LIN {X 0,Y 353.263,Z 401.913,A -85,B 0,C 180,E1 -13410,E2 -13410} C_VEL
LIN {X 0,Y 353.204,Z 401.841,A -85,B 0,C 180,E1 -13411.14,E2 -13411.14} C_VEL
LIN {X 0,Y 353.173,Z 401.369,A -85,B 0,C 180,E1 -13412.281,E2 -13412.281} C_VEL
LIN {X 0,Y 353.22,Z 400.459,A -85,B 0,C 180,E1 -13413.422,E2 -13413.422} C_VEL
LIN {X 0,Y 353.263,Z 399.147,A -85,B 0,C 180,E1 -13414.564,E2 -13414.564} C_VEL
LIN {X 0,Y 353.279,Z 397.099,A -85,B 0,C 180,E1 -13415.904,E2 -13415.904} C_VEL
LIN {X 0,Y 353.627,Z 392.597,A -85,B 0,C 180,E1 -13417.997,E2 -13417.997} C_VEL
LIN {X 0,Y 354.079,Z 387.694,A -85,B 0,C 180,E1 -13419.713,E2 -13419.713} C_VEL
LIN {X 0,Y 354.749,Z 381.546,A -85,B 0,C 180,E1 -13421.426,E2 -13421.426} C_VEL
LIN {X 0,Y 355.822,Z 373.938,A -85,B 0,C 180,E1 -13423.128,E2 -13423.128} C_VEL
LIN {X 0,Y 356.761,Z 366.198,A -85,B 0,C 180,E1 -13424.546,E2 -13424.546} C_VEL
LIN {X 0,Y 357.799,Z 356.811,A -85,B 0,C 180,E1 -13425.961,E2 -13425.961} C_VEL
LIN {X 0,Y 359.249,Z 345.191,A -85,B 0,C 180,E1 -13427.357,E2 -13427.357} C_VEL
LIN {X 0,Y 360.513,Z 333.695,A -85,B 0,C 180,E1 -13428.446,E2 -13428.446} C_VEL
LIN {X 0,Y 359.704,Z 322.357,A -85,B 0,C 180,E1 -13429.399,E2 -13429.399} C_VEL
LIN {X 0,Y 357.526,Z 309.013,A -85,B 0,C 180,E1 -13430.353,E2 -13430.353} C_VEL
LIN {X 0,Y 354.606,Z 296.916,A -85,B 0,C 180,E1 -13431.079,E2 -13431.079} C_VEL
LIN {X 0,Y 354.186,Z 294.731,A -85,B 0,C 180,E1 -13431.197,E2 -13431.197} C_VEL
LIN {X 0,Y 354.608,Z 288.932,A -85,B 0,C 180,E1 -13434.594,E2 -13434.594} C_VEL
LIN {X 0,Y 355.173,Z 282.758,A -85,B 0,C 180,E1 -13438.352,E2 -13438.352} C_VEL
LIN {X 0,Y 355.914,Z 276.694,A -85,B 0,C 180,E1 -13442.218,E2 -13442.218} C_VEL
LIN {X 0,Y 356.302,Z 272.736,A -85,B 0,C 180,E1 -13444.89,E2 -13444.89} C_VEL
LIN {X 0,Y 356.369,Z 270.793,A -85,B 0,C 180,E1 -13446.272,E2 -13446.272} C_VEL
LIN {X 0,Y 356.049,Z 266.987,A -85,B 0,C 180,E1 -13449.17,E2 -13449.17} C_VEL
LIN {X 0,Y 355.535,Z 263.321,A -85,B 0,C 180,E1 -13452.227,E2 -13452.227} C_VEL
LIN {X 0,Y 354.835,Z 259.51,A -85,B 0,C 180,E1 -13455.788,E2 -13455.788} C_VEL
LIN {X 0,Y 354.816,Z 259.293,A -85,B 0,C 180,E1 -13458.822,E2 -13458.822} C_VEL
LIN {X 0,Y 354.808,Z 259.292,A -85,B 0,C 180,E1 -13462.401,E2 -13462.401} C_VEL
LIN {X 0,Y 354.81,Z 259.29,A -85,B 0,C 180,E1 -13464.939,E2 -13464.939} C_VEL
LIN {X 0,Y 354.791,Z 259.293,A -85,B 0,C 180,E1 -13468.404,E2 -13468.404} C_VEL
LIN {X 0,Y 354.851,Z 259.284,A -85,B 0,C 180,E1 -13471.618,E2 -13471.618} C_VEL
LIN {X 0,Y 354.896,Z 259.28,A -85,B 0,C 180,E1 -13474.171,E2 -13474.171} C_VEL
LIN {X 0,Y 354.831,Z 259.288,A -85,B 0,C 180,E1 -13477.892,E2 -13477.892} C_VEL
LIN {X 0,Y 354.918,Z 259.277,A -85,B 0,C 180,E1 -13481.89,E2 -13481.89} C_VEL
LIN {X 0,Y 354.937,Z 259.275,A -85,B 0,C 180,E1 -13485.98,E2 -13485.98} C_VEL
LIN {X 0,Y 354.972,Z 259.27,A -85,B 0,C 180,E1 -13489.734,E2 -13489.734} C_VEL
LIN {X 0,Y 355.108,Z 259.254,A -85,B 0,C 180,E1 -13492.035,E2 -13492.035} C_VEL
LIN {X 0,Y 355.086,Z 259.255,A -85,B 0,C 180,E1 -13494.319,E2 -13494.319} C_VEL
LIN {X 0,Y 355.239,Z 259.237,A -85,B 0,C 180,E1 -13497.731,E2 -13497.731} C_VEL
LIN {X 0,Y 355.39,Z 259.217,A -85,B 0,C 180,E1 -13499.999,E2 -13499.999} C_VEL
LIN {X 0,Y 355.239,Z 259.238,A -85,B 0,C 180,E1 -13502.266,E2 -13502.266} C_VEL
LIN {X 0,Y 355.086,Z 259.257,A -85,B 0,C 180,E1 -13505.678,E2 -13505.678} C_VEL
LIN {X 0,Y 355.318,Z 260.942,A -85,B 0,C 180,E1 -13507.957,E2 -13507.957} C_VEL
LIN {X 0,Y 355.247,Z 264.154,A -85,B 0,C 180,E1 -13511.409,E2 -13511.409} C_VEL
LIN {X 0,Y 355.037,Z 266.823,A -85,B 0,C 180,E1 -13514.084,E2 -13514.084} C_VEL
LIN {X 0,Y 354.65,Z 270.896,A -85,B 0,C 180,E1 -13517.977,E2 -13517.977} C_VEL
LIN {X 0,Y 354.303,Z 274.435,A -85,B 0,C 180,E1 -13521.208,E2 -13521.208} C_VEL
LIN {X 0,Y 354.018,Z 278.57,A -85,B 0,C 180,E1 -13524.872,E2 -13524.872} C_VEL
LIN {X 0,Y 358.353,Z 293.464,A -85,B 0,C 180,E1 -13525.871,E2 -13525.871} C_VEL
LIN {X 0,Y 360.827,Z 304.889,A -85,B 0,C 180,E1 -13526.769,E2 -13526.769} C_VEL
LIN {X 0,Y 361.556,Z 309.621,A -85,B 0,C 180,E1 -13527.179,E2 -13527.179} C_VEL
LIN {X 0,Y 360.633,Z 320.768,A -85,B 0,C 180,E1 -13528.128,E2 -13528.128} C_VEL
LIN {X 0,Y 359.465,Z 331.353,A -85,B 0,C 180,E1 -13529.259,E2 -13529.259} C_VEL
LIN {X 0,Y 358.198,Z 341.935,A -85,B 0,C 180,E1 -13530.671,E2 -13530.671} C_VEL
LIN {X 0,Y 357.012,Z 351.025,A -85,B 0,C 180,E1 -13532.171,E2 -13532.171} C_VEL
LIN {X 0,Y 355.829,Z 359.612,A -85,B 0,C 180,E1 -13533.95,E2 -13533.95} C_VEL
LIN {X 0,Y 354.944,Z 366.442,A -85,B 0,C 180,E1 -13535.729,E2 -13535.729} C_VEL
LIN {X 0,Y 354.256,Z 371.77,A -85,B 0,C 180,E1 -13537.483,E2 -13537.483} C_VEL
LIN {X 0,Y 353.709,Z 376.354,A -85,B 0,C 180,E1 -13539.479,E2 -13539.479} C_VEL
LIN {X 0,Y 353.388,Z 378.94,A -85,B 0,C 180,E1 -13541.015,E2 -13541.015} C_VEL
LIN {X 0,Y 353.201,Z 380.756,A -85,B 0,C 180,E1 -13542.59,E2 -13542.59} C_VEL
LIN {X 0,Y 353.074,Z 381.837,A -85,B 0,C 180,E1 -13544.228,E2 -13544.228} C_VEL
LIN {X 0,Y 352.988,Z 382.113,A -85,B 0,C 180,E1 -13545.826,E2 -13545.826} C_VEL
LIN {X 0,Y 352.994,Z 381.593,A -85,B 0,C 180,E1 -13547.445,E2 -13547.445} C_VEL
LIN {X 0,Y 353.087,Z 380.151,A -85,B 0,C 180,E1 -13549.142,E2 -13549.142} C_VEL
LIN {X 0,Y 353.318,Z 377.739,A -85,B 0,C 180,E1 -13550.872,E2 -13550.872} C_VEL
LIN {X 0,Y 353.618,Z 374.206,A -85,B 0,C 180,E1 -13552.65,E2 -13552.65} C_VEL
LIN {X 0,Y 354.072,Z 369.386,A -85,B 0,C 180,E1 -13554.467,E2 -13554.467} C_VEL
LIN {X 0,Y 354.646,Z 362.944,A -85,B 0,C 180,E1 -13556.334,E2 -13556.334} C_VEL
LIN {X 0,Y 355.544,Z 354.73,A -85,B 0,C 180,E1 -13558.206,E2 -13558.206} C_VEL
LIN {X 0,Y 356.335,Z 346.798,A -85,B 0,C 180,E1 -13559.663,E2 -13559.663} C_VEL
LIN {X 0,Y 357.334,Z 336.482,A -85,B 0,C 180,E1 -13561.194,E2 -13561.194} C_VEL
LIN {X 0,Y 358.287,Z 326.115,A -85,B 0,C 180,E1 -13562.434,E2 -13562.434} C_VEL
LIN {X 0,Y 359.177,Z 315.981,A -85,B 0,C 180,E1 -13563.411,E2 -13563.411} C_VEL
LIN {X 0,Y 359.786,Z 307.654,A -85,B 0,C 180,E1 -13564.069,E2 -13564.069} C_VEL
LIN {X 0,Y 357.564,Z 294.986,A -85,B 0,C 180,E1 -13565.003,E2 -13565.003} C_VEL
LIN {X 0,Y 354.842,Z 282.519,A -85,B 0,C 180,E1 -13565.716,E2 -13565.716} C_VEL
LIN {X 0,Y 353.716,Z 277.507,A -85,B 0,C 180,E1 -13565.964,E2 -13565.964} C_VEL
LIN {X 0,Y 353.939,Z 273.668,A -85,B 0,C 180,E1 -13569.059,E2 -13569.059} C_VEL
LIN {X 0,Y 354.185,Z 269.276,A -85,B 0,C 180,E1 -13572.685,E2 -13572.685} C_VEL
LIN {X 0,Y 354.416,Z 264.974,A -85,B 0,C 180,E1 -13576.319,E2 -13576.319} C_VEL
LIN {X 0,Y 354.676,Z 261.044,A -85,B 0,C 180,E1 -13579.727,E2 -13579.727} C_VEL
LIN {X 0,Y 354.804,Z 259.289,A -85,B 0,C 180,E1 -13581.356,E2 -13581.356} C_VEL
LIN {X 0,Y 355.057,Z 259.257,A -85,B 0,C 180,E1 -13583.18,E2 -13583.18} C_VEL
LIN {X 0,Y 355.236,Z 259.233,A -85,B 0,C 180,E1 -13587.733,E2 -13587.733} C_VEL
LIN {X 0,Y 355.389,Z 259.215,A -85,B 0,C 180,E1 -13590,E2 -13590} C_VEL
LIN {X 0,Y 355.236,Z 259.237,A -85,B 0,C 180,E1 -13592.268,E2 -13592.268} C_VEL
LIN {X 0,Y 355.127,Z 259.248,A -85,B 0,C 180,E1 -13596.819,E2 -13596.819} C_VEL
LIN {X 0,Y 355.006,Z 259.262,A -85,B 0,C 180,E1 -13599.113,E2 -13599.113} C_VEL
LIN {X 0,Y 354.916,Z 259.275,A -85,B 0,C 180,E1 -13602.581,E2 -13602.581} C_VEL
LIN {X 0,Y 354.882,Z 259.282,A -85,B 0,C 180,E1 -13606.096,E2 -13606.096} C_VEL
LIN {X 0,Y 354.898,Z 259.277,A -85,B 0,C 180,E1 -13608.472,E2 -13608.472} C_VEL
LIN {X 0,Y 354.834,Z 259.288,A -85,B 0,C 180,E1 -13612.106,E2 -13612.106} C_VEL
LIN {X 0,Y 354.889,Z 259.281,A -85,B 0,C 180,E1 -13615.828,E2 -13615.828} C_VEL
LIN {X 0,Y 354.844,Z 259.286,A -85,B 0,C 180,E1 -13619.679,E2 -13619.679} C_VEL
LIN {X 0,Y 354.82,Z 259.29,A -85,B 0,C 180,E1 -13623.683,E2 -13623.683} C_VEL
LIN {X 0,Y 354.791,Z 259.288,A -85,B 0,C 180,E1 -13626.46,E2 -13626.46} C_VEL
LIN {X 0,Y 354.811,Z 259.29,A -85,B 0,C 180,E1 -13629.488,E2 -13629.488} C_VEL
LIN {X 0,Y 354.118,Z 259.373,A -85,B 0,C 180,E1 -13630.434,E2 -13630.434} C_VEL
LIN {X 0,Y 351.253,Z 259.73,A -85,B 0,C 180,E1 -13631.973,E2 -13631.973} C_VEL
LIN {X 0,Y 348.859,Z 260.031,A -85,B 0,C 180,E1 -13633.219,E2 -13633.219} C_VEL
LIN {X 0,Y 347.857,Z 260.152,A -85,B 0,C 180,E1 -13634.183,E2 -13634.183} C_VEL
LIN {X 0,Y 347.788,Z 260.16,A -85,B 0,C 180,E1 -13634.509,E2 -13634.509} C_VEL
LIN {X 0,Y 347.807,Z 260.159,A -85,B 0,C 180,E1 -13636.671,E2 -13636.671} C_VEL
LIN {X 0,Y 347.776,Z 260.162,A -85,B 0,C 180,E1 -13640.166,E2 -13640.166} C_VEL
LIN {X 0,Y 347.78,Z 260.161,A -85,B 0,C 180,E1 -13644.126,E2 -13644.126} C_VEL
LIN {X 0,Y 347.729,Z 260.168,A -85,B 0,C 180,E1 -13648.087,E2 -13648.087} C_VEL
LIN {X 0,Y 347.798,Z 260.165,A -85,B 0,C 180,E1 -13650.991,E2 -13650.991} C_VEL
LIN {X 0,Y 347.823,Z 260.157,A -85,B 0,C 180,E1 -13653.609,E2 -13653.609} C_VEL
LIN {X 0,Y 347.78,Z 260.162,A -85,B 0,C 180,E1 -13656.163,E2 -13656.163} C_VEL
LIN {X 0,Y 347.804,Z 260.158,A -85,B 0,C 180,E1 -13659.911,E2 -13659.911} C_VEL
LIN {X 0,Y 347.858,Z 260.155,A -85,B 0,C 180,E1 -13662.36,E2 -13662.36} C_VEL
LIN {X 0,Y 347.891,Z 260.148,A -85,B 0,C 180,E1 -13665.972,E2 -13665.972} C_VEL
LIN {X 0,Y 347.922,Z 260.144,A -85,B 0,C 180,E1 -13669.527,E2 -13669.527} C_VEL
LIN {X 0,Y 348.086,Z 260.124,A -85,B 0,C 180,E1 -13673.043,E2 -13673.043} C_VEL
LIN {X 0,Y 348.202,Z 260.11,A -85,B 0,C 180,E1 -13677.688,E2 -13677.688} C_VEL
LIN {X 0,Y 348.34,Z 260.095,A -85,B 0,C 180,E1 -13680.001,E2 -13680.001} C_VEL
LIN {X 0,Y 348.203,Z 260.113,A -85,B 0,C 180,E1 -13682.315,E2 -13682.315} C_VEL
LIN {X 0,Y 348.102,Z 260.122,A -85,B 0,C 180,E1 -13686.959,E2 -13686.959} C_VEL
LIN {X 0,Y 347.965,Z 260.139,A -85,B 0,C 180,E1 -13689.3,E2 -13689.3} C_VEL
LIN {X 0,Y 347.89,Z 260.148,A -85,B 0,C 180,E1 -13692.841,E2 -13692.841} C_VEL
LIN {X 0,Y 347.836,Z 260.155,A -85,B 0,C 180,E1 -13696.433,E2 -13696.433} C_VEL
LIN {X 0,Y 347.849,Z 260.153,A -85,B 0,C 180,E1 -13698.862,E2 -13698.862} C_VEL
LIN {X 0,Y 347.772,Z 260.163,A -85,B 0,C 180,E1 -13702.581,E2 -13702.581} C_VEL
LIN {X 0,Y 347.811,Z 260.159,A -85,B 0,C 180,E1 -13705.11,E2 -13705.11} C_VEL
LIN {X 0,Y 347.807,Z 260.163,A -85,B 0,C 180,E1 -13707.695,E2 -13707.695} C_VEL
LIN {X 0,Y 347.748,Z 260.165,A -85,B 0,C 180,E1 -13710.349,E2 -13710.349} C_VEL
LIN {X 0,Y 347.748,Z 260.166,A -85,B 0,C 180,E1 -13714.045,E2 -13714.045} C_VEL
LIN {X 0,Y 347.766,Z 260.168,A -85,B 0,C 180,E1 -13717.322,E2 -13717.322} C_VEL
LIN {X 0,Y 347.733,Z 260.167,A -85,B 0,C 180,E1 -13720.298,E2 -13720.298} C_VEL
LIN {X 0,Y 347.724,Z 260.172,A -85,B 0,C 180,E1 -13723.409,E2 -13723.409} C_VEL
LIN {X 0,Y 347.798,Z 260.25,A -85,B 0,C 180,E1 -13727.494,E2 -13727.494} C_VEL
LIN {X 0,Y 348.418,Z 263.797,A -85,B 0,C 180,E1 -13730.043,E2 -13730.043} C_VEL
LIN {X 0,Y 349.006,Z 267.844,A -85,B 0,C 180,E1 -13732.835,E2 -13732.835} C_VEL
LIN {X 0,Y 349.105,Z 271.117,A -85,B 0,C 180,E1 -13734.989,E2 -13734.989} C_VEL
LIN {X 0,Y 348.528,Z 276.532,A -85,B 0,C 180,E1 -13738.38,E2 -13738.38} C_VEL
LIN {X 0,Y 347.753,Z 283.788,A -85,B 0,C 180,E1 -13742.779,E2 -13742.779} C_VEL
LIN {X 0,Y 347.299,Z 289.444,A -85,B 0,C 180,E1 -13746.127,E2 -13746.127} C_VEL
LIN {X 0,Y 346.948,Z 295.615,A -85,B 0,C 180,E1 -13749.703,E2 -13749.703} C_VEL
LIN {X 0,Y 349.396,Z 309.468,A -85,B 0,C 180,E1 -13750.375,E2 -13750.375} C_VEL
LIN {X 0,Y 351.283,Z 322.744,A -85,B 0,C 180,E1 -13751.25,E2 -13751.25} C_VEL
LIN {X 0,Y 352.197,Z 331.78,A -85,B 0,C 180,E1 -13751.983,E2 -13751.983} C_VEL
LIN {X 0,Y 351.074,Z 344.156,A -85,B 0,C 180,E1 -13753.126,E2 -13753.126} C_VEL
LIN {X 0,Y 350.024,Z 354.445,A -85,B 0,C 180,E1 -13754.332,E2 -13754.332} C_VEL
LIN {X 0,Y 349.095,Z 364.017,A -85,B 0,C 180,E1 -13755.723,E2 -13755.723} C_VEL
LIN {X 0,Y 348.258,Z 372.23,A -85,B 0,C 180,E1 -13757.174,E2 -13757.174} C_VEL
LIN {X 0,Y 347.344,Z 380.282,A -85,B 0,C 180,E1 -13758.918,E2 -13758.918} C_VEL
LIN {X 0,Y 346.811,Z 386.74,A -85,B 0,C 180,E1 -13760.67,E2 -13760.67} C_VEL
LIN {X 0,Y 346.449,Z 391.853,A -85,B 0,C 180,E1 -13762.423,E2 -13762.423} C_VEL
LIN {X 0,Y 346.191,Z 396.427,A -85,B 0,C 180,E1 -13764.513,E2 -13764.513} C_VEL
LIN {X 0,Y 346.148,Z 399.438,A -85,B 0,C 180,E1 -13766.508,E2 -13766.508} C_VEL
LIN {X 0,Y 346.087,Z 400.627,A -85,B 0,C 180,E1 -13767.672,E2 -13767.672} C_VEL
LIN {X 0,Y 346.12,Z 401.366,A -85,B 0,C 180,E1 -13768.836,E2 -13768.836} C_VEL
LIN {X 0,Y 346.166,Z 401.703,A -85,B 0,C 180,E1 -13770,E2 -13770} C_VEL
LIN {X 0,Y 346.105,Z 401.646,A -85,B 0,C 180,E1 -13771.163,E2 -13771.163} C_VEL
LIN {X 0,Y 346.084,Z 401.195,A -85,B 0,C 180,E1 -13772.327,E2 -13772.327} C_VEL
LIN {X 0,Y 346.143,Z 400.303,A -85,B 0,C 180,E1 -13773.492,E2 -13773.492} C_VEL
LIN {X 0,Y 346.16,Z 399.003,A -85,B 0,C 180,E1 -13774.658,E2 -13774.658} C_VEL
LIN {X 0,Y 346.245,Z 396.272,A -85,B 0,C 180,E1 -13776.409,E2 -13776.409} C_VEL
LIN {X 0,Y 346.571,Z 392.525,A -85,B 0,C 180,E1 -13778.16,E2 -13778.16} C_VEL
LIN {X 0,Y 347.058,Z 387.668,A -85,B 0,C 180,E1 -13779.911,E2 -13779.911} C_VEL
LIN {X 0,Y 347.761,Z 381.564,A -85,B 0,C 180,E1 -13781.659,E2 -13781.659} C_VEL
LIN {X 0,Y 348.897,Z 374,A -85,B 0,C 180,E1 -13783.394,E2 -13783.394} C_VEL
LIN {X 0,Y 349.869,Z 366.316,A -85,B 0,C 180,E1 -13784.839,E2 -13784.839} C_VEL
LIN {X 0,Y 350.975,Z 357.024,A -85,B 0,C 180,E1 -13786.28,E2 -13786.28} C_VEL
LIN {X 0,Y 352.294,Z 346.766,A -85,B 0,C 180,E1 -13787.561,E2 -13787.561} C_VEL
LIN {X 0,Y 353.687,Z 335.617,A -85,B 0,C 180,E1 -13788.676,E2 -13788.676} C_VEL
LIN {X 0,Y 353.468,Z 327.837,A -85,B 0,C 180,E1 -13789.384,E2 -13789.384} C_VEL
LIN {X 0,Y 352.13,Z 316.947,A -85,B 0,C 180,E1 -13790.271,E2 -13790.271} C_VEL
LIN {X 0,Y 349.593,Z 304.104,A -85,B 0,C 180,E1 -13791.158,E2 -13791.158} C_VEL
LIN {X 0,Y 347.218,Z 294.508,A -85,B 0,C 180,E1 -13791.734,E2 -13791.734} C_VEL
LIN {X 0,Y 347.721,Z 287.86,A -85,B 0,C 180,E1 -13795.756,E2 -13795.756} C_VEL
LIN {X 0,Y 348.389,Z 281.407,A -85,B 0,C 180,E1 -13799.836,E2 -13799.836} C_VEL
LIN {X 0,Y 348.988,Z 276.74,A -85,B 0,C 180,E1 -13802.937,E2 -13802.937} C_VEL
LIN {X 0,Y 349.338,Z 272.82,A -85,B 0,C 180,E1 -13805.691,E2 -13805.691} C_VEL
LIN {X 0,Y 349.151,Z 269.001,A -85,B 0,C 180,E1 -13808.607,E2 -13808.607} C_VEL
LIN {X 0,Y 348.64,Z 265.244,A -85,B 0,C 180,E1 -13811.766,E2 -13811.766} C_VEL
LIN {X 0,Y 348.05,Z 261.753,A -85,B 0,C 180,E1 -13815.028,E2 -13815.028} C_VEL
LIN {X 0,Y 347.732,Z 260.172,A -85,B 0,C 180,E1 -13816.684,E2 -13816.684} C_VEL
LIN {X 0,Y 347.757,Z 260.171,A -85,B 0,C 180,E1 -13820.169,E2 -13820.169} C_VEL
LIN {X 0,Y 347.77,Z 260.167,A -85,B 0,C 180,E1 -13823.933,E2 -13823.933} C_VEL
LIN {X 0,Y 347.731,Z 260.173,A -85,B 0,C 180,E1 -13826.926,E2 -13826.926} C_VEL
LIN {X 0,Y 347.804,Z 260.162,A -85,B 0,C 180,E1 -13830.989,E2 -13830.989} C_VEL
LIN {X 0,Y 347.829,Z 260.159,A -85,B 0,C 180,E1 -13833.606,E2 -13833.606} C_VEL
LIN {X 0,Y 347.785,Z 260.164,A -85,B 0,C 180,E1 -13836.16,E2 -13836.16} C_VEL
LIN {X 0,Y 347.808,Z 260.162,A -85,B 0,C 180,E1 -13839.908,E2 -13839.908} C_VEL
LIN {X 0,Y 347.862,Z 260.155,A -85,B 0,C 180,E1 -13842.358,E2 -13842.358} C_VEL
LIN {X 0,Y 347.893,Z 260.152,A -85,B 0,C 180,E1 -13845.969,E2 -13845.969} C_VEL
LIN {X 0,Y 347.923,Z 260.148,A -85,B 0,C 180,E1 -13849.524,E2 -13849.524} C_VEL
LIN {X 0,Y 348.068,Z 260.13,A -85,B 0,C 180,E1 -13851.873,E2 -13851.873} C_VEL
LIN {X 0,Y 348.061,Z 260.131,A -85,B 0,C 180,E1 -13854.204,E2 -13854.204} C_VEL
LIN {X 0,Y 348.201,Z 260.114,A -85,B 0,C 180,E1 -13857.685,E2 -13857.685} C_VEL
LIN {X 0,Y 348.339,Z 260.095,A -85,B 0,C 180,E1 -13859.999,E2 -13859.999} C_VEL
LIN {X 0,Y 348.201,Z 260.115,A -85,B 0,C 180,E1 -13862.312,E2 -13862.312} C_VEL
LIN {X 0,Y 348.067,Z 260.363,A -85,B 0,C 180,E1 -13865.793,E2 -13865.793} C_VEL
LIN {X 0,Y 348.344,Z 262.793,A -85,B 0,C 180,E1 -13868.669,E2 -13868.669} C_VEL
LIN {X 0,Y 348.209,Z 265.53,A -85,B 0,C 180,E1 -13871.643,E2 -13871.643} C_VEL
LIN {X 0,Y 347.996,Z 268.045,A -85,B 0,C 180,E1 -13874.218,E2 -13874.218} C_VEL
LIN {X 0,Y 347.588,Z 272.064,A -85,B 0,C 180,E1 -13878.142,E2 -13878.142} C_VEL
LIN {X 0,Y 347.241,Z 275.581,A -85,B 0,C 180,E1 -13881.409,E2 -13881.409} C_VEL
LIN {X 0,Y 347.012,Z 278.831,A -85,B 0,C 180,E1 -13884.347,E2 -13884.347} C_VEL
LIN {X 0,Y 351.254,Z 292.936,A -85,B 0,C 180,E1 -13885.319,E2 -13885.319} C_VEL
LIN {X 0,Y 353.8,Z 304.235,A -85,B 0,C 180,E1 -13886.229,E2 -13886.229} C_VEL
LIN {X 0,Y 354.878,Z 310.676,A -85,B 0,C 180,E1 -13886.809,E2 -13886.809} C_VEL
LIN {X 0,Y 353.887,Z 321.994,A -85,B 0,C 180,E1 -13887.818,E2 -13887.818} C_VEL
LIN {X 0,Y 352.504,Z 333.902,A -85,B 0,C 180,E1 -13889.162,E2 -13889.162} C_VEL
LIN {X 0,Y 351.162,Z 344.174,A -85,B 0,C 180,E1 -13890.62,E2 -13890.62} C_VEL
LIN {X 0,Y 349.936,Z 353.033,A -85,B 0,C 180,E1 -13892.187,E2 -13892.187} C_VEL
LIN {X 0,Y 348.782,Z 360.872,A -85,B 0,C 180,E1 -13893.898,E2 -13893.898} C_VEL
LIN {X 0,Y 347.814,Z 367.989,A -85,B 0,C 180,E1 -13895.87,E2 -13895.87} C_VEL
LIN {X 0,Y 347.072,Z 373.448,A -85,B 0,C 180,E1 -13897.842,E2 -13897.842} C_VEL
LIN {X 0,Y 346.584,Z 377.122,A -85,B 0,C 180,E1 -13899.597,E2 -13899.597} C_VEL
LIN {X 0,Y 346.25,Z 379.739,A -85,B 0,C 180,E1 -13901.324,E2 -13901.324} C_VEL
LIN {X 0,Y 345.994,Z 381.851,A -85,B 0,C 180,E1 -13903.677,E2 -13903.677} C_VEL
LIN {X 0,Y 345.904,Z 382.317,A -85,B 0,C 180,E1 -13905.324,E2 -13905.324} C_VEL
LIN {X 0,Y 345.876,Z 381.98,A -85,B 0,C 180,E1 -13907.009,E2 -13907.009} C_VEL
LIN {X 0,Y 345.949,Z 380.771,A -85,B 0,C 180,E1 -13908.732,E2 -13908.732} C_VEL
LIN {X 0,Y 346.244,Z 377.798,A -85,B 0,C 180,E1 -13911.008,E2 -13911.008} C_VEL
LIN {X 0,Y 346.516,Z 374.856,A -85,B 0,C 180,E1 -13912.523,E2 -13912.523} C_VEL
LIN {X 0,Y 346.913,Z 370.872,A -85,B 0,C 180,E1 -13914.127,E2 -13914.127} C_VEL
LIN {X 0,Y 347.459,Z 364.861,A -85,B 0,C 180,E1 -13916.024,E2 -13916.024} C_VEL
LIN {X 0,Y 348.191,Z 357.957,A -85,B 0,C 180,E1 -13917.75,E2 -13917.75} C_VEL
LIN {X 0,Y 349.112,Z 349.448,A -85,B 0,C 180,E1 -13919.45,E2 -13919.45} C_VEL
LIN {X 0,Y 350.068,Z 339.648,A -85,B 0,C 180,E1 -13921.032,E2 -13921.032} C_VEL
LIN {X 0,Y 351.114,Z 329.663,A -85,B 0,C 180,E1 -13922.331,E2 -13922.331} C_VEL
LIN {X 0,Y 352.066,Z 319.164,A -85,B 0,C 180,E1 -13923.431,E2 -13923.431} C_VEL
LIN {X 0,Y 352.868,Z 308.463,A -85,B 0,C 180,E1 -13924.331,E2 -13924.331} C_VEL
LIN {X 0,Y 350.654,Z 295.841,A -85,B 0,C 180,E1 -13925.294,E2 -13925.294} C_VEL
LIN {X 0,Y 347.953,Z 283.457,A -85,B 0,C 180,E1 -13926.033,E2 -13926.033} C_VEL
LIN {X 0,Y 346.66,Z 277.682,A -85,B 0,C 180,E1 -13926.318,E2 -13926.318} C_VEL
LIN {X 0,Y 346.888,Z 273.399,A -85,B 0,C 180,E1 -13929.854,E2 -13929.854} C_VEL
LIN {X 0,Y 347.147,Z 269.032,A -85,B 0,C 180,E1 -13933.535,E2 -13933.535} C_VEL
LIN {X 0,Y 347.447,Z 264.848,A -85,B 0,C 180,E1 -13937.144,E2 -13937.144} C_VEL
LIN {X 0,Y 347.701,Z 260.85,A -85,B 0,C 180,E1 -13940.695,E2 -13940.695} C_VEL
LIN {X 0,Y 347.805,Z 260.159,A -85,B 0,C 180,E1 -13941.576,E2 -13941.576} C_VEL
LIN {X 0,Y 348.036,Z 260.131,A -85,B 0,C 180,E1 -13944.205,E2 -13944.205} C_VEL
LIN {X 0,Y 348.198,Z 260.109,A -85,B 0,C 180,E1 -13947.687,E2 -13947.687} C_VEL
LIN {X 0,Y 348.358,Z 260.091,A -85,B 0,C 180,E1 -13950,E2 -13950} C_VEL
LIN {X 0,Y 348.198,Z 260.113,A -85,B 0,C 180,E1 -13952.314,E2 -13952.314} C_VEL
LIN {X 0,Y 348.096,Z 260.123,A -85,B 0,C 180,E1 -13956.958,E2 -13956.958} C_VEL
LIN {X 0,Y 347.959,Z 260.139,A -85,B 0,C 180,E1 -13959.299,E2 -13959.299} C_VEL
LIN {X 0,Y 347.884,Z 260.149,A -85,B 0,C 180,E1 -13962.84,E2 -13962.84} C_VEL
LIN {X 0,Y 347.831,Z 260.158,A -85,B 0,C 180,E1 -13966.432,E2 -13966.432} C_VEL
LIN {X 0,Y 347.849,Z 260.153,A -85,B 0,C 180,E1 -13968.86,E2 -13968.86} C_VEL
LIN {X 0,Y 347.771,Z 260.163,A -85,B 0,C 180,E1 -13972.579,E2 -13972.579} C_VEL
LIN {X 0,Y 347.807,Z 260.158,A -85,B 0,C 180,E1 -13975.109,E2 -13975.109} C_VEL
LIN {X 0,Y 347.802,Z 260.163,A -85,B 0,C 180,E1 -13977.694,E2 -13977.694} C_VEL
LIN {X 0,Y 347.76,Z 260.165,A -85,B 0,C 180,E1 -13980.346,E2 -13980.346} C_VEL
LIN {X 0,Y 347.738,Z 260.169,A -85,B 0,C 180,E1 -13984.044,E2 -13984.044} C_VEL
LIN {X 0,Y 347.756,Z 260.168,A -85,B 0,C 180,E1 -13987.321,E2 -13987.321} C_VEL
LIN {X 0,Y 347.783,Z 260.161,A -85,B 0,C 180,E1 -13990.289,E2 -13990.289} C_VEL
LIN {X 0,Y 347.809,Z 260.163,A -85,B 0,C 180,E1 -13993.394,E2 -13993.394} C_VEL
LIN {X 0,Y 347.788,Z 260.16,A -85,B 0,C 180,E1 -13994.509,E2 -13994.509} C_VEL
LIN {X 0,Y 347.14,Z 260.246,A -85,B 0,C 180,E1 -13995.476,E2 -13995.476} C_VEL
LIN {X 0,Y 344.249,Z 260.604,A -85,B 0,C 180,E1 -13997.048,E2 -13997.048} C_VEL
LIN {X 0,Y 341.81,Z 260.905,A -85,B 0,C 180,E1 -13998.322,E2 -13998.322} C_VEL
LIN {X 0,Y 340.804,Z 261.036,A -85,B 0,C 180,E1 -13999.308,E2 -13999.308} C_VEL
LIN {X 0,Y 340.746,Z 261.039,A -85,B 0,C 180,E1 -13999.641,E2 -13999.641} C_VEL
LIN {X 0,Y 340.696,Z 261.049,A -85,B 0,C 180,E1 -14003.26,E2 -14003.26} C_VEL
LIN {X 0,Y 340.683,Z 261.045,A -85,B 0,C 180,E1 -14006.154,E2 -14006.154} C_VEL
LIN {X 0,Y 340.766,Z 261.036,A -85,B 0,C 180,E1 -14010.334,E2 -14010.334} C_VEL
LIN {X 0,Y 340.797,Z 261.036,A -85,B 0,C 180,E1 -14013.021,E2 -14013.021} C_VEL
LIN {X 0,Y 340.72,Z 261.046,A -85,B 0,C 180,E1 -14016.928,E2 -14016.928} C_VEL
LIN {X 0,Y 340.783,Z 261.038,A -85,B 0,C 180,E1 -14020.735,E2 -14020.735} C_VEL
LIN {X 0,Y 340.779,Z 261.035,A -85,B 0,C 180,E1 -14023.22,E2 -14023.22} C_VEL
LIN {X 0,Y 340.837,Z 261.029,A -85,B 0,C 180,E1 -14026.892,E2 -14026.892} C_VEL
LIN {X 0,Y 340.907,Z 261.023,A -85,B 0,C 180,E1 -14030.509,E2 -14030.509} C_VEL
LIN {X 0,Y 341.053,Z 261.001,A -85,B 0,C 180,E1 -14032.899,E2 -14032.899} C_VEL
LIN {X 0,Y 341.164,Z 260.986,A -85,B 0,C 180,E1 -14037.64,E2 -14037.64} C_VEL
LIN {X 0,Y 341.291,Z 260.973,A -85,B 0,C 180,E1 -14040.001,E2 -14040.001} C_VEL
LIN {X 0,Y 341.165,Z 260.989,A -85,B 0,C 180,E1 -14042.363,E2 -14042.363} C_VEL
LIN {X 0,Y 341.071,Z 260.997,A -85,B 0,C 180,E1 -14047.103,E2 -14047.103} C_VEL
LIN {X 0,Y 340.871,Z 261.022,A -85,B 0,C 180,E1 -14050.695,E2 -14050.695} C_VEL
LIN {X 0,Y 340.86,Z 261.025,A -85,B 0,C 180,E1 -14054.326,E2 -14054.326} C_VEL
LIN {X 0,Y 340.835,Z 261.027,A -85,B 0,C 180,E1 -14058.468,E2 -14058.468} C_VEL
LIN {X 0,Y 340.752,Z 261.041,A -85,B 0,C 180,E1 -14061.858,E2 -14061.858} C_VEL
LIN {X 0,Y 340.771,Z 261.039,A -85,B 0,C 180,E1 -14065.666,E2 -14065.666} C_VEL
LIN {X 0,Y 340.727,Z 261.04,A -85,B 0,C 180,E1 -14068.322,E2 -14068.322} C_VEL
LIN {X 0,Y 340.697,Z 261.046,A -85,B 0,C 180,E1 -14071.046,E2 -14071.046} C_VEL
LIN {X 0,Y 340.718,Z 261.046,A -85,B 0,C 180,E1 -14075.28,E2 -14075.28} C_VEL
LIN {X 0,Y 340.712,Z 261.042,A -85,B 0,C 180,E1 -14078.388,E2 -14078.388} C_VEL
LIN {X 0,Y 340.7,Z 261.043,A -85,B 0,C 180,E1 -14082.047,E2 -14082.047} C_VEL
LIN {X 0,Y 340.655,Z 261.054,A -85,B 0,C 180,E1 -14086.228,E2 -14086.228} C_VEL
LIN {X 0,Y 340.76,Z 261.239,A -85,B 0,C 180,E1 -14087.356,E2 -14087.356} C_VEL
LIN {X 0,Y 341.476,Z 265.342,A -85,B 0,C 180,E1 -14090.357,E2 -14090.357} C_VEL
LIN {X 0,Y 342.025,Z 269.739,A -85,B 0,C 180,E1 -14093.424,E2 -14093.424} C_VEL
LIN {X 0,Y 342.044,Z 272.527,A -85,B 0,C 180,E1 -14095.275,E2 -14095.275} C_VEL
LIN {X 0,Y 341.34,Z 278.413,A -85,B 0,C 180,E1 -14099.021,E2 -14099.021} C_VEL
LIN {X 0,Y 340.656,Z 284.871,A -85,B 0,C 180,E1 -14103.008,E2 -14103.008} C_VEL
LIN {X 0,Y 340.214,Z 290.224,A -85,B 0,C 180,E1 -14106.246,E2 -14106.246} C_VEL
LIN {X 0,Y 339.913,Z 295.409,A -85,B 0,C 180,E1 -14109.32,E2 -14109.32} C_VEL
LIN {X 0,Y 342.631,Z 310.98,A -85,B 0,C 180,E1 -14110.13,E2 -14110.13} C_VEL
LIN {X 0,Y 344.269,Z 322.784,A -85,B 0,C 180,E1 -14110.936,E2 -14110.936} C_VEL
LIN {X 0,Y 345.288,Z 332.642,A -85,B 0,C 180,E1 -14111.764,E2 -14111.764} C_VEL
LIN {X 0,Y 344.1,Z 344.785,A -85,B 0,C 180,E1 -14112.927,E2 -14112.927} C_VEL
LIN {X 0,Y 342.956,Z 355.539,A -85,B 0,C 180,E1 -14114.245,E2 -14114.245} C_VEL
LIN {X 0,Y 341.972,Z 365.259,A -85,B 0,C 180,E1 -14115.723,E2 -14115.723} C_VEL
LIN {X 0,Y 341.107,Z 373.236,A -85,B 0,C 180,E1 -14117.204,E2 -14117.204} C_VEL
LIN {X 0,Y 340.241,Z 381.036,A -85,B 0,C 180,E1 -14118.985,E2 -14118.985} C_VEL
LIN {X 0,Y 339.618,Z 388.198,A -85,B 0,C 180,E1 -14121.071,E2 -14121.071} C_VEL
LIN {X 0,Y 339.274,Z 392.956,A -85,B 0,C 180,E1 -14122.86,E2 -14122.86} C_VEL
LIN {X 0,Y 339.14,Z 395.607,A -85,B 0,C 180,E1 -14124.108,E2 -14124.108} C_VEL
LIN {X 0,Y 339.077,Z 397.549,A -85,B 0,C 180,E1 -14125.244,E2 -14125.244} C_VEL
LIN {X 0,Y 339.072,Z 399.17,A -85,B 0,C 180,E1 -14126.435,E2 -14126.435} C_VEL
LIN {X 0,Y 339.002,Z 400.377,A -85,B 0,C 180,E1 -14127.624,E2 -14127.624} C_VEL
LIN {X 0,Y 339.022,Z 401.141,A -85,B 0,C 180,E1 -14128.812,E2 -14128.812} C_VEL
LIN {X 0,Y 339.069,Z 401.493,A -85,B 0,C 180,E1 -14130,E2 -14130} C_VEL
LIN {X 0,Y 339.008,Z 401.451,A -85,B 0,C 180,E1 -14131.188,E2 -14131.188} C_VEL
LIN {X 0,Y 338.999,Z 401.019,A -85,B 0,C 180,E1 -14132.376,E2 -14132.376} C_VEL
LIN {X 0,Y 339.067,Z 400.157,A -85,B 0,C 180,E1 -14133.565,E2 -14133.565} C_VEL
LIN {X 0,Y 339.115,Z 397.341,A -85,B 0,C 180,E1 -14135.849,E2 -14135.849} C_VEL
LIN {X 0,Y 339.404,Z 393.819,A -85,B 0,C 180,E1 -14137.735,E2 -14137.735} C_VEL
LIN {X 0,Y 339.853,Z 389.382,A -85,B 0,C 180,E1 -14139.522,E2 -14139.522} C_VEL
LIN {X 0,Y 340.55,Z 383.76,A -85,B 0,C 180,E1 -14141.306,E2 -14141.306} C_VEL
LIN {X 0,Y 341.566,Z 376.773,A -85,B 0,C 180,E1 -14143.081,E2 -14143.081} C_VEL
LIN {X 0,Y 342.815,Z 368.062,A -85,B 0,C 180,E1 -14144.848,E2 -14144.848} C_VEL
LIN {X 0,Y 343.876,Z 359.381,A -85,B 0,C 180,E1 -14146.296,E2 -14146.296} C_VEL
LIN {X 0,Y 345.394,Z 348.413,A -85,B 0,C 180,E1 -14147.771,E2 -14147.771} C_VEL
LIN {X 0,Y 346.856,Z 337.594,A -85,B 0,C 180,E1 -14148.916,E2 -14148.916} C_VEL
LIN {X 0,Y 346.954,Z 331.795,A -85,B 0,C 180,E1 -14149.472,E2 -14149.472} C_VEL
LIN {X 0,Y 345.866,Z 320.781,A -85,B 0,C 180,E1 -14150.449,E2 -14150.449} C_VEL
LIN {X 0,Y 343.682,Z 308.315,A -85,B 0,C 180,E1 -14151.396,E2 -14151.396} C_VEL
LIN {X 0,Y 340.219,Z 294.271,A -85,B 0,C 180,E1 -14152.314,E2 -14152.314} C_VEL
LIN {X 0,Y 340.736,Z 287.831,A -85,B 0,C 180,E1 -14156.324,E2 -14156.324} C_VEL
LIN {X 0,Y 341.418,Z 281.929,A -85,B 0,C 180,E1 -14160.166,E2 -14160.166} C_VEL
LIN {X 0,Y 341.923,Z 278.39,A -85,B 0,C 180,E1 -14162.569,E2 -14162.569} C_VEL
LIN {X 0,Y 342.276,Z 274.842,A -85,B 0,C 180,E1 -14165.094,E2 -14165.094} C_VEL
LIN {X 0,Y 342.342,Z 272.551,A -85,B 0,C 180,E1 -14166.807,E2 -14166.807} C_VEL
LIN {X 0,Y 342.016,Z 269.14,A -85,B 0,C 180,E1 -14169.568,E2 -14169.568} C_VEL
LIN {X 0,Y 341.477,Z 265.519,A -85,B 0,C 180,E1 -14172.778,E2 -14172.778} C_VEL
LIN {X 0,Y 340.873,Z 262.096,A -85,B 0,C 180,E1 -14176.187,E2 -14176.187} C_VEL
LIN {X 0,Y 340.703,Z 261.049,A -85,B 0,C 180,E1 -14177.575,E2 -14177.575} C_VEL
LIN {X 0,Y 340.709,Z 261.049,A -85,B 0,C 180,E1 -14180.247,E2 -14180.247} C_VEL
LIN {X 0,Y 340.709,Z 261.048,A -85,B 0,C 180,E1 -14183.558,E2 -14183.558} C_VEL
LIN {X 0,Y 340.69,Z 261.049,A -85,B 0,C 180,E1 -14186.152,E2 -14186.152} C_VEL
LIN {X 0,Y 340.773,Z 261.038,A -85,B 0,C 180,E1 -14190.331,E2 -14190.331} C_VEL
LIN {X 0,Y 340.802,Z 261.035,A -85,B 0,C 180,E1 -14193.019,E2 -14193.019} C_VEL
LIN {X 0,Y 340.725,Z 261.045,A -85,B 0,C 180,E1 -14196.926,E2 -14196.926} C_VEL
LIN {X 0,Y 340.786,Z 261.037,A -85,B 0,C 180,E1 -14200.732,E2 -14200.732} C_VEL
LIN {X 0,Y 340.782,Z 261.039,A -85,B 0,C 180,E1 -14203.217,E2 -14203.217} C_VEL
LIN {X 0,Y 340.839,Z 261.03,A -85,B 0,C 180,E1 -14206.889,E2 -14206.889} C_VEL
LIN {X 0,Y 340.923,Z 261.021,A -85,B 0,C 180,E1 -14210.506,E2 -14210.506} C_VEL
LIN {X 0,Y 341.069,Z 261.002,A -85,B 0,C 180,E1 -14212.897,E2 -14212.897} C_VEL
LIN {X 0,Y 341.163,Z 260.991,A -85,B 0,C 180,E1 -14217.637,E2 -14217.637} C_VEL
LIN {X 0,Y 341.289,Z 260.973,A -85,B 0,C 180,E1 -14219.999,E2 -14219.999} C_VEL
LIN {X 0,Y 341.163,Z 260.991,A -85,B 0,C 180,E1 -14222.36,E2 -14222.36} C_VEL
LIN {X 0,Y 340.84,Z 261.033,A -85,B 0,C 180,E1 -14224.73,E2 -14224.73} C_VEL
LIN {X 0,Y 341.237,Z 262.681,A -85,B 0,C 180,E1 -14227.097,E2 -14227.097} C_VEL
LIN {X 0,Y 341.291,Z 264.729,A -85,B 0,C 180,E1 -14229.481,E2 -14229.481} C_VEL
LIN {X 0,Y 341.16,Z 266.908,A -85,B 0,C 180,E1 -14231.887,E2 -14231.887} C_VEL
LIN {X 0,Y 340.948,Z 269.27,A -85,B 0,C 180,E1 -14234.351,E2 -14234.351} C_VEL
LIN {X 0,Y 340.593,Z 272.952,A -85,B 0,C 180,E1 -14238.029,E2 -14238.029} C_VEL
LIN {X 0,Y 340.132,Z 276.961,A -85,B 0,C 180,E1 -14241.833,E2 -14241.833} C_VEL
LIN {X 0,Y 339.993,Z 279.053,A -85,B 0,C 180,E1 -14243.769,E2 -14243.769} C_VEL
LIN {X 0,Y 344.11,Z 292.507,A -85,B 0,C 180,E1 -14244.742,E2 -14244.742} C_VEL
LIN {X 0,Y 346.971,Z 304.354,A -85,B 0,C 180,E1 -14245.734,E2 -14245.734} C_VEL
LIN {X 0,Y 348.269,Z 312.731,A -85,B 0,C 180,E1 -14246.516,E2 -14246.516} C_VEL
LIN {X 0,Y 347.052,Z 324.212,A -85,B 0,C 180,E1 -14247.593,E2 -14247.593} C_VEL
LIN {X 0,Y 345.819,Z 334.144,A -85,B 0,C 180,E1 -14248.756,E2 -14248.756} C_VEL
LIN {X 0,Y 344.516,Z 343.847,A -85,B 0,C 180,E1 -14250.153,E2 -14250.153} C_VEL
LIN {X 0,Y 343.404,Z 351.389,A -85,B 0,C 180,E1 -14251.472,E2 -14251.472} C_VEL
LIN {X 0,Y 342.181,Z 359.338,A -85,B 0,C 180,E1 -14253.166,E2 -14253.166} C_VEL
LIN {X 0,Y 341.199,Z 365.751,A -85,B 0,C 180,E1 -14254.849,E2 -14254.849} C_VEL
LIN {X 0,Y 340.354,Z 371.594,A -85,B 0,C 180,E1 -14256.784,E2 -14256.784} C_VEL
LIN {X 0,Y 339.835,Z 375.295,A -85,B 0,C 180,E1 -14258.344,E2 -14258.344} C_VEL
LIN {X 0,Y 339.258,Z 379.418,A -85,B 0,C 180,E1 -14260.731,E2 -14260.731} C_VEL
LIN {X 0,Y 339.107,Z 380.632,A -85,B 0,C 180,E1 -14261.748,E2 -14261.748} C_VEL
LIN {X 0,Y 338.923,Z 381.996,A -85,B 0,C 180,E1 -14263.469,E2 -14263.469} C_VEL
LIN {X 0,Y 338.828,Z 382.511,A -85,B 0,C 180,E1 -14265.153,E2 -14265.153} C_VEL
LIN {X 0,Y 338.782,Z 382.255,A -85,B 0,C 180,E1 -14266.799,E2 -14266.799} C_VEL
LIN {X 0,Y 338.85,Z 381.271,A -85,B 0,C 180,E1 -14268.418,E2 -14268.418} C_VEL
LIN {X 0,Y 339.123,Z 378.334,A -85,B 0,C 180,E1 -14270.831,E2 -14270.831} C_VEL
LIN {X 0,Y 339.424,Z 375.243,A -85,B 0,C 180,E1 -14272.509,E2 -14272.509} C_VEL
LIN {X 0,Y 339.945,Z 369.984,A -85,B 0,C 180,E1 -14274.63,E2 -14274.63} C_VEL
LIN {X 0,Y 340.527,Z 363.92,A -85,B 0,C 180,E1 -14276.491,E2 -14276.491} C_VEL
LIN {X 0,Y 341.443,Z 356.153,A -85,B 0,C 180,E1 -14278.368,E2 -14278.368} C_VEL
LIN {X 0,Y 342.265,Z 348.483,A -85,B 0,C 180,E1 -14279.874,E2 -14279.874} C_VEL
LIN {X 0,Y 343.243,Z 338.941,A -85,B 0,C 180,E1 -14281.413,E2 -14281.413} C_VEL
LIN {X 0,Y 344.383,Z 327.86,A -85,B 0,C 180,E1 -14282.832,E2 -14282.832} C_VEL
LIN {X 0,Y 345.536,Z 315.637,A -85,B 0,C 180,E1 -14284.069,E2 -14284.069} C_VEL
LIN {X 0,Y 345.971,Z 309.366,A -85,B 0,C 180,E1 -14284.588,E2 -14284.588} C_VEL
LIN {X 0,Y 343.694,Z 296.296,A -85,B 0,C 180,E1 -14285.613,E2 -14285.613} C_VEL
LIN {X 0,Y 340.968,Z 283.81,A -85,B 0,C 180,E1 -14286.382,E2 -14286.382} C_VEL
LIN {X 0,Y 339.613,Z 277.874,A -85,B 0,C 180,E1 -14286.686,E2 -14286.686} C_VEL
LIN {X 0,Y 339.794,Z 274.615,A -85,B 0,C 180,E1 -14289.415,E2 -14289.415} C_VEL
LIN {X 0,Y 340.059,Z 270.207,A -85,B 0,C 180,E1 -14293.182,E2 -14293.182} C_VEL
LIN {X 0,Y 340.386,Z 265.981,A -85,B 0,C 180,E1 -14296.873,E2 -14296.873} C_VEL
LIN {X 0,Y 340.648,Z 261.961,A -85,B 0,C 180,E1 -14300.5,E2 -14300.5} C_VEL
LIN {X 0,Y 340.732,Z 261.041,A -85,B 0,C 180,E1 -14301.4,E2 -14301.4} C_VEL
LIN {X 0,Y 341.007,Z 261.006,A -85,B 0,C 180,E1 -14304.086,E2 -14304.086} C_VEL
LIN {X 0,Y 341.16,Z 260.986,A -85,B 0,C 180,E1 -14307.639,E2 -14307.639} C_VEL
LIN {X 0,Y 341.307,Z 260.969,A -85,B 0,C 180,E1 -14310,E2 -14310} C_VEL
LIN {X 0,Y 341.16,Z 260.99,A -85,B 0,C 180,E1 -14312.361,E2 -14312.361} C_VEL
LIN {X 0,Y 341.065,Z 260.998,A -85,B 0,C 180,E1 -14317.102,E2 -14317.102} C_VEL
LIN {X 0,Y 340.865,Z 261.025,A -85,B 0,C 180,E1 -14320.694,E2 -14320.694} C_VEL
LIN {X 0,Y 340.852,Z 261.029,A -85,B 0,C 180,E1 -14324.325,E2 -14324.325} C_VEL
LIN {X 0,Y 340.828,Z 261.03,A -85,B 0,C 180,E1 -14328.468,E2 -14328.468} C_VEL
LIN {X 0,Y 340.743,Z 261.042,A -85,B 0,C 180,E1 -14331.857,E2 -14331.857} C_VEL
LIN {X 0,Y 340.765,Z 261.039,A -85,B 0,C 180,E1 -14335.665,E2 -14335.665} C_VEL
LIN {X 0,Y 340.732,Z 261.041,A -85,B 0,C 180,E1 -14338.32,E2 -14338.32} C_VEL
LIN {X 0,Y 340.705,Z 261.043,A -85,B 0,C 180,E1 -14341.043,E2 -14341.043} C_VEL
LIN {X 0,Y 340.708,Z 261.045,A -85,B 0,C 180,E1 -14345.279,E2 -14345.279} C_VEL
LIN {X 0,Y 340.709,Z 261.042,A -85,B 0,C 180,E1 -14348.389,E2 -14348.389} C_VEL
LIN {X 0,Y 340.716,Z 261.045,A -85,B 0,C 180,E1 -14351.304,E2 -14351.304} C_VEL
LIN {X 0,Y 340.771,Z 261.034,A -85,B 0,C 180,E1 -14354.523,E2 -14354.523} C_VEL
LIN {X 0,Y 340.742,Z 261.039,A -85,B 0,C 180,E1 -14357.946,E2 -14357.946} C_VEL
LIN {X 0,Y 340.746,Z 261.039,A -85,B 0,C 180,E1 -14359.641,E2 -14359.641} C_VEL
LIN {X 0,Y 340.125,Z 261.119,A -85,B 0,C 180,E1 -14360.628,E2 -14360.628} C_VEL
LIN {X 0,Y 337.236,Z 261.476,A -85,B 0,C 180,E1 -14362.232,E2 -14362.232} C_VEL
LIN {X 0,Y 334.767,Z 261.785,A -85,B 0,C 180,E1 -14363.531,E2 -14363.531} C_VEL
LIN {X 0,Y 333.727,Z 261.912,A -85,B 0,C 180,E1 -14364.538,E2 -14364.538} C_VEL
LIN {X 0,Y 333.656,Z 261.922,A -85,B 0,C 180,E1 -14364.879,E2 -14364.879} C_VEL
LIN {X 0,Y 333.624,Z 261.925,A -85,B 0,C 180,E1 -14368.223,E2 -14368.223} C_VEL
LIN {X 0,Y 333.703,Z 261.92,A -85,B 0,C 180,E1 -14371.029,E2 -14371.029} C_VEL
LIN {X 0,Y 333.728,Z 261.912,A -85,B 0,C 180,E1 -14373.755,E2 -14373.755} C_VEL
LIN {X 0,Y 333.712,Z 261.914,A -85,B 0,C 180,E1 -14377.915,E2 -14377.915} C_VEL
LIN {X 0,Y 333.786,Z 261.904,A -85,B 0,C 180,E1 -14381.591,E2 -14381.591} C_VEL
LIN {X 0,Y 333.801,Z 261.902,A -85,B 0,C 180,E1 -14385.578,E2 -14385.578} C_VEL
LIN {X 0,Y 333.827,Z 261.9,A -85,B 0,C 180,E1 -14389.079,E2 -14389.079} C_VEL
LIN {X 0,Y 334,Z 261.88,A -85,B 0,C 180,E1 -14392.748,E2 -14392.748} C_VEL
LIN {X 0,Y 333.804,Z 261.902,A -85,B 0,C 180,E1 -14395.17,E2 -14395.17} C_VEL
LIN {X 0,Y 334.101,Z 261.866,A -85,B 0,C 180,E1 -14397.59,E2 -14397.59} C_VEL
LIN {X 0,Y 334.242,Z 261.851,A -85,B 0,C 180,E1 -14400.001,E2 -14400.001} C_VEL
LIN {X 0,Y 334.102,Z 261.868,A -85,B 0,C 180,E1 -14402.413,E2 -14402.413} C_VEL
LIN {X 0,Y 334.021,Z 261.875,A -85,B 0,C 180,E1 -14407.254,E2 -14407.254} C_VEL
LIN {X 0,Y 333.834,Z 261.898,A -85,B 0,C 180,E1 -14410.923,E2 -14410.923} C_VEL
LIN {X 0,Y 333.806,Z 261.902,A -85,B 0,C 180,E1 -14414.636,E2 -14414.636} C_VEL
LIN {X 0,Y 333.794,Z 261.903,A -85,B 0,C 180,E1 -14418.656,E2 -14418.656} C_VEL
LIN {X 0,Y 333.691,Z 261.917,A -85,B 0,C 180,E1 -14422.28,E2 -14422.28} C_VEL
LIN {X 0,Y 333.734,Z 261.911,A -85,B 0,C 180,E1 -14426.248,E2 -14426.248} C_VEL
LIN {X 0,Y 333.689,Z 261.918,A -85,B 0,C 180,E1 -14428.975,E2 -14428.975} C_VEL
LIN {X 0,Y 333.643,Z 261.922,A -85,B 0,C 180,E1 -14432.588,E2 -14432.588} C_VEL
LIN {X 0,Y 333.677,Z 261.918,A -85,B 0,C 180,E1 -14436.14,E2 -14436.14} C_VEL
LIN {X 0,Y 333.648,Z 261.927,A -85,B 0,C 180,E1 -14439.194,E2 -14439.194} C_VEL
LIN {X 0,Y 333.633,Z 261.924,A -85,B 0,C 180,E1 -14442.501,E2 -14442.501} C_VEL
LIN {X 0,Y 333.7,Z 262.025,A -85,B 0,C 180,E1 -14447.068,E2 -14447.068} C_VEL
LIN {X 0,Y 334.585,Z 267.228,A -85,B 0,C 180,E1 -14450.939,E2 -14450.939} C_VEL
LIN {X 0,Y 335.035,Z 271.62,A -85,B 0,C 180,E1 -14454.031,E2 -14454.031} C_VEL
LIN {X 0,Y 334.86,Z 274.881,A -85,B 0,C 180,E1 -14456.209,E2 -14456.209} C_VEL
LIN {X 0,Y 334.153,Z 280.267,A -85,B 0,C 180,E1 -14459.684,E2 -14459.684} C_VEL
LIN {X 0,Y 333.421,Z 287.794,A -85,B 0,C 180,E1 -14464.4,E2 -14464.4} C_VEL
LIN {X 0,Y 332.87,Z 295.193,A -85,B 0,C 180,E1 -14468.912,E2 -14468.912} C_VEL
LIN {X 0,Y 332.872,Z 295.315,A -85,B 0,C 180,E1 -14468.966,E2 -14468.966} C_VEL
LIN {X 0,Y 335.271,Z 308.852,A -85,B 0,C 180,E1 -14469.65,E2 -14469.65} C_VEL
LIN {X 0,Y 337.279,Z 322.519,A -85,B 0,C 180,E1 -14470.595,E2 -14470.595} C_VEL
LIN {X 0,Y 338.368,Z 333.378,A -85,B 0,C 180,E1 -14471.534,E2 -14471.534} C_VEL
LIN {X 0,Y 337.13,Z 345.274,A -85,B 0,C 180,E1 -14472.719,E2 -14472.719} C_VEL
LIN {X 0,Y 335.956,Z 355.91,A -85,B 0,C 180,E1 -14474.064,E2 -14474.064} C_VEL
LIN {X 0,Y 335.064,Z 364.643,A -85,B 0,C 180,E1 -14475.422,E2 -14475.422} C_VEL
LIN {X 0,Y 334.166,Z 372.691,A -85,B 0,C 180,E1 -14476.933,E2 -14476.933} C_VEL
LIN {X 0,Y 333.211,Z 380.574,A -85,B 0,C 180,E1 -14478.75,E2 -14478.75} C_VEL
LIN {X 0,Y 332.749,Z 385.934,A -85,B 0,C 180,E1 -14480.272,E2 -14480.272} C_VEL
LIN {X 0,Y 332.323,Z 391.148,A -85,B 0,C 180,E1 -14482.099,E2 -14482.099} C_VEL
LIN {X 0,Y 332.065,Z 395.536,A -85,B 0,C 180,E1 -14484.125,E2 -14484.125} C_VEL
LIN {X 0,Y 331.998,Z 398.888,A -85,B 0,C 180,E1 -14486.359,E2 -14486.359} C_VEL
LIN {X 0,Y 331.919,Z 400.114,A -85,B 0,C 180,E1 -14487.573,E2 -14487.573} C_VEL
LIN {X 0,Y 331.927,Z 400.913,A -85,B 0,C 180,E1 -14488.787,E2 -14488.787} C_VEL
LIN {X 0,Y 331.972,Z 401.283,A -85,B 0,C 180,E1 -14490,E2 -14490} C_VEL
LIN {X 0,Y 331.916,Z 400.842,A -85,B 0,C 180,E1 -14492.427,E2 -14492.427} C_VEL
LIN {X 0,Y 331.97,Z 400.013,A -85,B 0,C 180,E1 -14493.641,E2 -14493.641} C_VEL
LIN {X 0,Y 332.009,Z 397.523,A -85,B 0,C 180,E1 -14495.78,E2 -14495.78} C_VEL
LIN {X 0,Y 332.361,Z 393.742,A -85,B 0,C 180,E1 -14497.9,E2 -14497.9} C_VEL
LIN {X 0,Y 332.823,Z 389.34,A -85,B 0,C 180,E1 -14499.725,E2 -14499.725} C_VEL
LIN {X 0,Y 333.559,Z 383.77,A -85,B 0,C 180,E1 -14501.546,E2 -14501.546} C_VEL
LIN {X 0,Y 334.639,Z 376.853,A -85,B 0,C 180,E1 -14503.357,E2 -14503.357} C_VEL
LIN {X 0,Y 335.941,Z 368.252,A -85,B 0,C 180,E1 -14505.159,E2 -14505.159} C_VEL
LIN {X 0,Y 337.014,Z 360.01,A -85,B 0,C 180,E1 -14506.579,E2 -14506.579} C_VEL
LIN {X 0,Y 338.497,Z 349.94,A -85,B 0,C 180,E1 -14507.989,E2 -14507.989} C_VEL
LIN {X 0,Y 340.01,Z 339.589,A -85,B 0,C 180,E1 -14509.155,E2 -14509.155} C_VEL
LIN {X 0,Y 340.316,Z 333.953,A -85,B 0,C 180,E1 -14509.723,E2 -14509.723} C_VEL
LIN {X 0,Y 339.4,Z 323.195,A -85,B 0,C 180,E1 -14510.74,E2 -14510.74} C_VEL
LIN {X 0,Y 337.468,Z 311.359,A -85,B 0,C 180,E1 -14511.714,E2 -14511.714} C_VEL
LIN {X 0,Y 334.321,Z 298.354,A -85,B 0,C 180,E1 -14512.63,E2 -14512.63} C_VEL
LIN {X 0,Y 333.211,Z 294.101,A -85,B 0,C 180,E1 -14512.887,E2 -14512.887} C_VEL
LIN {X 0,Y 333.78,Z 287.82,A -85,B 0,C 180,E1 -14516.916,E2 -14516.916} C_VEL
LIN {X 0,Y 334.456,Z 282.453,A -85,B 0,C 180,E1 -14520.508,E2 -14520.508} C_VEL
LIN {X 0,Y 334.972,Z 278.814,A -85,B 0,C 180,E1 -14523.058,E2 -14523.058} C_VEL
LIN {X 0,Y 335.311,Z 274.927,A -85,B 0,C 180,E1 -14525.934,E2 -14525.934} C_VEL
LIN {X 0,Y 335.305,Z 273.03,A -85,B 0,C 180,E1 -14527.432,E2 -14527.432} C_VEL
LIN {X 0,Y 334.902,Z 269.325,A -85,B 0,C 180,E1 -14530.581,E2 -14530.581} C_VEL
LIN {X 0,Y 334.281,Z 265.335,A -85,B 0,C 180,E1 -14534.37,E2 -14534.37} C_VEL
LIN {X 0,Y 333.701,Z 261.932,A -85,B 0,C 180,E1 -14538.033,E2 -14538.033} C_VEL
LIN {X 0,Y 333.677,Z 261.924,A -85,B 0,C 180,E1 -14541.195,E2 -14541.195} C_VEL
LIN {X 0,Y 333.684,Z 261.921,A -85,B 0,C 180,E1 -14545.224,E2 -14545.224} C_VEL
LIN {X 0,Y 333.695,Z 261.92,A -85,B 0,C 180,E1 -14549.636,E2 -14549.636} C_VEL
LIN {X 0,Y 333.742,Z 261.913,A -85,B 0,C 180,E1 -14552.4,E2 -14552.4} C_VEL
LIN {X 0,Y 333.723,Z 261.916,A -85,B 0,C 180,E1 -14555.089,E2 -14555.089} C_VEL
LIN {X 0,Y 333.676,Z 261.922,A -85,B 0,C 180,E1 -14559.018,E2 -14559.018} C_VEL
LIN {X 0,Y 333.789,Z 261.908,A -85,B 0,C 180,E1 -14561.588,E2 -14561.588} C_VEL
LIN {X 0,Y 333.804,Z 261.907,A -85,B 0,C 180,E1 -14565.575,E2 -14565.575} C_VEL
LIN {X 0,Y 333.828,Z 261.903,A -85,B 0,C 180,E1 -14569.077,E2 -14569.077} C_VEL
LIN {X 0,Y 334.019,Z 261.881,A -85,B 0,C 180,E1 -14572.746,E2 -14572.746} C_VEL
LIN {X 0,Y 333.805,Z 261.904,A -85,B 0,C 180,E1 -14575.168,E2 -14575.168} C_VEL
LIN {X 0,Y 334.101,Z 261.871,A -85,B 0,C 180,E1 -14577.587,E2 -14577.587} C_VEL
LIN {X 0,Y 334.24,Z 261.851,A -85,B 0,C 180,E1 -14579.999,E2 -14579.999} C_VEL
LIN {X 0,Y 334.1,Z 261.871,A -85,B 0,C 180,E1 -14582.41,E2 -14582.41} C_VEL
LIN {X 0,Y 333.848,Z 262.237,A -85,B 0,C 180,E1 -14584.829,E2 -14584.829} C_VEL
LIN {X 0,Y 334.257,Z 264.068,A -85,B 0,C 180,E1 -14587.246,E2 -14587.246} C_VEL
LIN {X 0,Y 334.292,Z 266.106,A -85,B 0,C 180,E1 -14589.681,E2 -14589.681} C_VEL
LIN {X 0,Y 334.114,Z 268.308,A -85,B 0,C 180,E1 -14592.141,E2 -14592.141} C_VEL
LIN {X 0,Y 333.742,Z 271.848,A -85,B 0,C 180,E1 -14595.886,E2 -14595.886} C_VEL
LIN {X 0,Y 333.309,Z 275.701,A -85,B 0,C 180,E1 -14599.715,E2 -14599.715} C_VEL
LIN {X 0,Y 333.01,Z 279.483,A -85,B 0,C 180,E1 -14603.185,E2 -14603.185} C_VEL
LIN {X 0,Y 337.276,Z 292.597,A -85,B 0,C 180,E1 -14604.177,E2 -14604.177} C_VEL
LIN {X 0,Y 340.139,Z 304.57,A -85,B 0,C 180,E1 -14605.219,E2 -14605.219} C_VEL
LIN {X 0,Y 341.609,Z 313.432,A -85,B 0,C 180,E1 -14606.086,E2 -14606.086} C_VEL
LIN {X 0,Y 340.515,Z 324.087,A -85,B 0,C 180,E1 -14607.111,E2 -14607.111} C_VEL
LIN {X 0,Y 339.03,Z 335.459,A -85,B 0,C 180,E1 -14608.474,E2 -14608.474} C_VEL
LIN {X 0,Y 337.566,Z 345.391,A -85,B 0,C 180,E1 -14609.976,E2 -14609.976} C_VEL
LIN {X 0,Y 336.292,Z 353.573,A -85,B 0,C 180,E1 -14611.496,E2 -14611.496} C_VEL
LIN {X 0,Y 334.922,Z 361.967,A -85,B 0,C 180,E1 -14613.422,E2 -14613.422} C_VEL
LIN {X 0,Y 333.837,Z 368.874,A -85,B 0,C 180,E1 -14615.467,E2 -14615.467} C_VEL
LIN {X 0,Y 333.135,Z 373.474,A -85,B 0,C 180,E1 -14617.197,E2 -14617.197} C_VEL
LIN {X 0,Y 332.506,Z 377.803,A -85,B 0,C 180,E1 -14619.35,E2 -14619.35} C_VEL
LIN {X 0,Y 332.115,Z 380.153,A -85,B 0,C 180,E1 -14620.993,E2 -14620.993} C_VEL
LIN {X 0,Y 331.923,Z 381.758,A -85,B 0,C 180,E1 -14622.65,E2 -14622.65} C_VEL
LIN {X 0,Y 331.758,Z 382.61,A -85,B 0,C 180,E1 -14624.35,E2 -14624.35} C_VEL
LIN {X 0,Y 331.708,Z 382.653,A -85,B 0,C 180,E1 -14626.082,E2 -14626.082} C_VEL
LIN {X 0,Y 331.688,Z 381.859,A -85,B 0,C 180,E1 -14627.865,E2 -14627.865} C_VEL
LIN {X 0,Y 331.847,Z 380.16,A -85,B 0,C 180,E1 -14629.675,E2 -14629.675} C_VEL
LIN {X 0,Y 332.156,Z 377.458,A -85,B 0,C 180,E1 -14631.521,E2 -14631.521} C_VEL
LIN {X 0,Y 332.621,Z 372.844,A -85,B 0,C 180,E1 -14633.729,E2 -14633.729} C_VEL
LIN {X 0,Y 333.191,Z 367.216,A -85,B 0,C 180,E1 -14635.731,E2 -14635.731} C_VEL
LIN {X 0,Y 334.03,Z 359.536,A -85,B 0,C 180,E1 -14637.825,E2 -14637.825} C_VEL
LIN {X 0,Y 334.983,Z 351.482,A -85,B 0,C 180,E1 -14639.572,E2 -14639.572} C_VEL
LIN {X 0,Y 336.044,Z 341.843,A -85,B 0,C 180,E1 -14641.249,E2 -14641.249} C_VEL
LIN {X 0,Y 337.169,Z 331.422,A -85,B 0,C 180,E1 -14642.706,E2 -14642.706} C_VEL
LIN {X 0,Y 338.327,Z 320.034,A -85,B 0,C 180,E1 -14643.975,E2 -14643.975} C_VEL
LIN {X 0,Y 339.068,Z 310.208,A -85,B 0,C 180,E1 -14644.856,E2 -14644.856} C_VEL
LIN {X 0,Y 336.987,Z 298.184,A -85,B 0,C 180,E1 -14645.841,E2 -14645.841} C_VEL
LIN {X 0,Y 334.06,Z 284.51,A -85,B 0,C 180,E1 -14646.727,E2 -14646.727} C_VEL
LIN {X 0,Y 332.553,Z 278.05,A -85,B 0,C 180,E1 -14647.068,E2 -14647.068} C_VEL
LIN {X 0,Y 332.759,Z 274.337,A -85,B 0,C 180,E1 -14650.25,E2 -14650.25} C_VEL
LIN {X 0,Y 332.972,Z 271.387,A -85,B 0,C 180,E1 -14652.813,E2 -14652.813} C_VEL
LIN {X 0,Y 333.289,Z 267.125,A -85,B 0,C 180,E1 -14656.588,E2 -14656.588} C_VEL
LIN {X 0,Y 333.585,Z 263.075,A -85,B 0,C 180,E1 -14660.297,E2 -14660.297} C_VEL
LIN {X 0,Y 333.717,Z 261.915,A -85,B 0,C 180,E1 -14661.523,E2 -14661.523} C_VEL
LIN {X 0,Y 333.975,Z 261.881,A -85,B 0,C 180,E1 -14663.961,E2 -14663.961} C_VEL
LIN {X 0,Y 334.097,Z 261.866,A -85,B 0,C 180,E1 -14667.589,E2 -14667.589} C_VEL
LIN {X 0,Y 334.257,Z 261.847,A -85,B 0,C 180,E1 -14670,E2 -14670} C_VEL
LIN {X 0,Y 334.121,Z 261.868,A -85,B 0,C 180,E1 -14672.411,E2 -14672.411} C_VEL
LIN {X 0,Y 334.015,Z 261.876,A -85,B 0,C 180,E1 -14677.253,E2 -14677.253} C_VEL
LIN {X 0,Y 333.827,Z 261.9,A -85,B 0,C 180,E1 -14680.922,E2 -14680.922} C_VEL
LIN {X 0,Y 333.798,Z 261.905,A -85,B 0,C 180,E1 -14684.635,E2 -14684.635} C_VEL
LIN {X 0,Y 333.787,Z 261.905,A -85,B 0,C 180,E1 -14688.656,E2 -14688.656} C_VEL
LIN {X 0,Y 333.684,Z 261.92,A -85,B 0,C 180,E1 -14692.279,E2 -14692.279} C_VEL
LIN {X 0,Y 333.727,Z 261.914,A -85,B 0,C 180,E1 -14696.247,E2 -14696.247} C_VEL
LIN {X 0,Y 333.701,Z 261.915,A -85,B 0,C 180,E1 -14698.973,E2 -14698.973} C_VEL
LIN {X 0,Y 333.641,Z 261.922,A -85,B 0,C 180,E1 -14702.59,E2 -14702.59} C_VEL
LIN {X 0,Y 333.667,Z 261.92,A -85,B 0,C 180,E1 -14706.139,E2 -14706.139} C_VEL
LIN {X 0,Y 333.675,Z 261.921,A -85,B 0,C 180,E1 -14709.188,E2 -14709.188} C_VEL
LIN {X 0,Y 333.693,Z 261.916,A -85,B 0,C 180,E1 -14712.514,E2 -14712.514} C_VEL
LIN {X 0,Y 333.719,Z 261.914,A -85,B 0,C 180,E1 -14715.978,E2 -14715.978} C_VEL
LIN {X 0,Y 333.669,Z 261.921,A -85,B 0,C 180,E1 -14719.63,E2 -14719.63} C_VEL
LIN {X 0,Y 333.656,Z 261.926,A -85,B 0,C 180,E1 -14723.169,E2 -14723.169} C_VEL
LIN {X 0,Y 333.656,Z 261.922,A -85,B 0,C 180,E1 -14724.879,E2 -14724.879} C_VEL
LIN {X 0,Y 333.015,Z 262.007,A -85,B 0,C 180,E1 -14725.885,E2 -14725.885} C_VEL
LIN {X 0,Y 330.146,Z 262.363,A -85,B 0,C 180,E1 -14727.522,E2 -14727.522} C_VEL
LIN {X 0,Y 327.719,Z 262.664,A -85,B 0,C 180,E1 -14728.848,E2 -14728.848} C_VEL
LIN {X 0,Y 326.709,Z 262.786,A -85,B 0,C 180,E1 -14729.875,E2 -14729.875} C_VEL
LIN {X 0,Y 326.645,Z 262.794,A -85,B 0,C 180,E1 -14730.223,E2 -14730.223} C_VEL
LIN {X 0,Y 326.677,Z 262.793,A -85,B 0,C 180,E1 -14733.144,E2 -14733.144} C_VEL
LIN {X 0,Y 326.644,Z 262.794,A -85,B 0,C 180,E1 -14735.872,E2 -14735.872} C_VEL
LIN {X 0,Y 326.658,Z 262.792,A -85,B 0,C 180,E1 -14739.866,E2 -14739.866} C_VEL
LIN {X 0,Y 326.692,Z 262.791,A -85,B 0,C 180,E1 -14742.473,E2 -14742.473} C_VEL
LIN {X 0,Y 326.752,Z 262.783,A -85,B 0,C 180,E1 -14746.316,E2 -14746.316} C_VEL
LIN {X 0,Y 326.8,Z 262.776,A -85,B 0,C 180,E1 -14750.095,E2 -14750.095} C_VEL
LIN {X 0,Y 326.984,Z 262.753,A -85,B 0,C 180,E1 -14753.832,E2 -14753.832} C_VEL
LIN {X 0,Y 327.042,Z 262.744,A -85,B 0,C 180,E1 -14757.538,E2 -14757.538} C_VEL
LIN {X 0,Y 327.193,Z 262.729,A -85,B 0,C 180,E1 -14760.001,E2 -14760.001} C_VEL
LIN {X 0,Y 327.043,Z 262.747,A -85,B 0,C 180,E1 -14762.465,E2 -14762.465} C_VEL
LIN {X 0,Y 326.992,Z 262.755,A -85,B 0,C 180,E1 -14766.171,E2 -14766.171} C_VEL
LIN {X 0,Y 326.912,Z 262.761,A -85,B 0,C 180,E1 -14768.657,E2 -14768.657} C_VEL
LIN {X 0,Y 326.735,Z 262.784,A -85,B 0,C 180,E1 -14772.423,E2 -14772.423} C_VEL
LIN {X 0,Y 326.752,Z 262.78,A -85,B 0,C 180,E1 -14774.959,E2 -14774.959} C_VEL
LIN {X 0,Y 326.731,Z 262.783,A -85,B 0,C 180,E1 -14778.839,E2 -14778.839} C_VEL
LIN {X 0,Y 326.62,Z 262.797,A -85,B 0,C 180,E1 -14782.789,E2 -14782.789} C_VEL
LIN {X 0,Y 326.689,Z 262.793,A -85,B 0,C 180,E1 -14785.485,E2 -14785.485} C_VEL
LIN {X 0,Y 326.647,Z 262.797,A -85,B 0,C 180,E1 -14789.662,E2 -14789.662} C_VEL
LIN {X 0,Y 326.607,Z 262.799,A -85,B 0,C 180,E1 -14794.021,E2 -14794.021} C_VEL
LIN {X 0,Y 326.63,Z 262.801,A -85,B 0,C 180,E1 -14797.24,E2 -14797.24} C_VEL
LIN {X 0,Y 326.579,Z 262.807,A -85,B 0,C 180,E1 -14801.133,E2 -14801.133} C_VEL
LIN {X 0,Y 326.529,Z 262.811,A -85,B 0,C 180,E1 -14804.744,E2 -14804.744} C_VEL
LIN {X 0,Y 326.622,Z 262.849,A -85,B 0,C 180,E1 -14806.8,E2 -14806.8} C_VEL
LIN {X 0,Y 327.367,Z 266.893,A -85,B 0,C 180,E1 -14809.906,E2 -14809.906} C_VEL
LIN {X 0,Y 327.909,Z 271.302,A -85,B 0,C 180,E1 -14813.122,E2 -14813.122} C_VEL
LIN {X 0,Y 327.924,Z 274.582,A -85,B 0,C 180,E1 -14815.394,E2 -14815.394} C_VEL
LIN {X 0,Y 327.164,Z 280.372,A -85,B 0,C 180,E1 -14819.236,E2 -14819.236} C_VEL
LIN {X 0,Y 326.414,Z 287.487,A -85,B 0,C 180,E1 -14823.808,E2 -14823.808} C_VEL
LIN {X 0,Y 325.904,Z 294.202,A -85,B 0,C 180,E1 -14828.017,E2 -14828.017} C_VEL
LIN {X 0,Y 325.834,Z 295.091,A -85,B 0,C 180,E1 -14828.568,E2 -14828.568} C_VEL
LIN {X 0,Y 328.256,Z 308.565,A -85,B 0,C 180,E1 -14829.268,E2 -14829.268} C_VEL
LIN {X 0,Y 330.151,Z 321.239,A -85,B 0,C 180,E1 -14830.159,E2 -14830.159} C_VEL
LIN {X 0,Y 331.294,Z 332.525,A -85,B 0,C 180,E1 -14831.143,E2 -14831.143} C_VEL
LIN {X 0,Y 331.152,Z 337.263,A -85,B 0,C 180,E1 -14831.598,E2 -14831.598} C_VEL
LIN {X 0,Y 329.879,Z 348.328,A -85,B 0,C 180,E1 -14832.806,E2 -14832.806} C_VEL
LIN {X 0,Y 328.766,Z 358.145,A -85,B 0,C 180,E1 -14834.149,E2 -14834.149} C_VEL
LIN {X 0,Y 327.719,Z 367.457,A -85,B 0,C 180,E1 -14835.723,E2 -14835.723} C_VEL
LIN {X 0,Y 326.682,Z 376.344,A -85,B 0,C 180,E1 -14837.577,E2 -14837.577} C_VEL
LIN {X 0,Y 325.901,Z 383.464,A -85,B 0,C 180,E1 -14839.438,E2 -14839.438} C_VEL
LIN {X 0,Y 325.379,Z 389.138,A -85,B 0,C 180,E1 -14841.304,E2 -14841.304} C_VEL
LIN {X 0,Y 325.058,Z 393.591,A -85,B 0,C 180,E1 -14843.171,E2 -14843.171} C_VEL
LIN {X 0,Y 324.899,Z 396.945,A -85,B 0,C 180,E1 -14845.036,E2 -14845.036} C_VEL
LIN {X 0,Y 324.902,Z 398.605,A -85,B 0,C 180,E1 -14846.279,E2 -14846.279} C_VEL
LIN {X 0,Y 324.84,Z 399.85,A -85,B 0,C 180,E1 -14847.52,E2 -14847.52} C_VEL
LIN {X 0,Y 324.836,Z 400.682,A -85,B 0,C 180,E1 -14848.76,E2 -14848.76} C_VEL
LIN {X 0,Y 324.876,Z 401.072,A -85,B 0,C 180,E1 -14850,E2 -14850} C_VEL
LIN {X 0,Y 324.836,Z 400.665,A -85,B 0,C 180,E1 -14852.48,E2 -14852.48} C_VEL
LIN {X 0,Y 324.877,Z 399.866,A -85,B 0,C 180,E1 -14853.721,E2 -14853.721} C_VEL
LIN {X 0,Y 324.912,Z 397.686,A -85,B 0,C 180,E1 -14855.723,E2 -14855.723} C_VEL
LIN {X 0,Y 325.292,Z 393.681,A -85,B 0,C 180,E1 -14858.073,E2 -14858.073} C_VEL
LIN {X 0,Y 325.808,Z 389.333,A -85,B 0,C 180,E1 -14859.937,E2 -14859.937} C_VEL
LIN {X 0,Y 326.7,Z 382.794,A -85,B 0,C 180,E1 -14862.107,E2 -14862.107} C_VEL
LIN {X 0,Y 327.973,Z 375.658,A -85,B 0,C 180,E1 -14863.949,E2 -14863.949} C_VEL
LIN {X 0,Y 329.265,Z 366.819,A -85,B 0,C 180,E1 -14865.791,E2 -14865.791} C_VEL
LIN {X 0,Y 330.741,Z 356.838,A -85,B 0,C 180,E1 -14867.466,E2 -14867.466} C_VEL
LIN {X 0,Y 332.517,Z 345.457,A -85,B 0,C 180,E1 -14868.963,E2 -14868.963} C_VEL
LIN {X 0,Y 333.675,Z 335.983,A -85,B 0,C 180,E1 -14869.984,E2 -14869.984} C_VEL
LIN {X 0,Y 332.948,Z 325.668,A -85,B 0,C 180,E1 -14871.029,E2 -14871.029} C_VEL
LIN {X 0,Y 331.279,Z 314.351,A -85,B 0,C 180,E1 -14872.03,E2 -14872.03} C_VEL
LIN {X 0,Y 328.355,Z 301.482,A -85,B 0,C 180,E1 -14873.019,E2 -14873.019} C_VEL
LIN {X 0,Y 326.224,Z 293.846,A -85,B 0,C 180,E1 -14873.538,E2 -14873.538} C_VEL
LIN {X 0,Y 326.853,Z 287.82,A -85,B 0,C 180,E1 -14877.526,E2 -14877.526} C_VEL
LIN {X 0,Y 327.506,Z 282.805,A -85,B 0,C 180,E1 -14880.998,E2 -14880.998} C_VEL
LIN {X 0,Y 328.05,Z 278.881,A -85,B 0,C 180,E1 -14883.848,E2 -14883.848} C_VEL
LIN {X 0,Y 328.293,Z 276.625,A -85,B 0,C 180,E1 -14885.56,E2 -14885.56} C_VEL
LIN {X 0,Y 328.199,Z 273.157,A -85,B 0,C 180,E1 -14888.388,E2 -14888.388} C_VEL
LIN {X 0,Y 327.734,Z 269.5,A -85,B 0,C 180,E1 -14891.663,E2 -14891.663} C_VEL
LIN {X 0,Y 327.176,Z 266.04,A -85,B 0,C 180,E1 -14895.141,E2 -14895.141} C_VEL
LIN {X 0,Y 326.61,Z 262.807,A -85,B 0,C 180,E1 -14898.861,E2 -14898.861} C_VEL
LIN {X 0,Y 326.642,Z 262.801,A -85,B 0,C 180,E1 -14901.393,E2 -14901.393} C_VEL
LIN {X 0,Y 326.618,Z 262.802,A -85,B 0,C 180,E1 -14904.85,E2 -14904.85} C_VEL
LIN {X 0,Y 326.606,Z 262.803,A -85,B 0,C 180,E1 -14907.454,E2 -14907.454} C_VEL
LIN {X 0,Y 326.659,Z 262.796,A -85,B 0,C 180,E1 -14910.339,E2 -14910.339} C_VEL
LIN {X 0,Y 326.687,Z 262.793,A -85,B 0,C 180,E1 -14914.515,E2 -14914.515} C_VEL
LIN {X 0,Y 326.642,Z 262.798,A -85,B 0,C 180,E1 -14918.544,E2 -14918.544} C_VEL
LIN {X 0,Y 326.741,Z 262.786,A -85,B 0,C 180,E1 -14921.176,E2 -14921.176} C_VEL
LIN {X 0,Y 326.758,Z 262.784,A -85,B 0,C 180,E1 -14925.432,E2 -14925.432} C_VEL
LIN {X 0,Y 326.765,Z 262.783,A -85,B 0,C 180,E1 -14928.837,E2 -14928.837} C_VEL
LIN {X 0,Y 326.973,Z 262.758,A -85,B 0,C 180,E1 -14932.589,E2 -14932.589} C_VEL
LIN {X 0,Y 326.772,Z 262.78,A -85,B 0,C 180,E1 -14935.063,E2 -14935.063} C_VEL
LIN {X 0,Y 327.041,Z 262.75,A -85,B 0,C 180,E1 -14937.535,E2 -14937.535} C_VEL
LIN {X 0,Y 327.191,Z 262.729,A -85,B 0,C 180,E1 -14939.999,E2 -14939.999} C_VEL
LIN {X 0,Y 327.041,Z 262.75,A -85,B 0,C 180,E1 -14942.462,E2 -14942.462} C_VEL
LIN {X 0,Y 326.791,Z 262.783,A -85,B 0,C 180,E1 -14943.698,E2 -14943.698} C_VEL
LIN {X 0,Y 327.276,Z 265.462,A -85,B 0,C 180,E1 -14947.401,E2 -14947.401} C_VEL
LIN {X 0,Y 327.277,Z 267.494,A -85,B 0,C 180,E1 -14949.891,E2 -14949.891} C_VEL
LIN {X 0,Y 327.081,Z 269.703,A -85,B 0,C 180,E1 -14952.406,E2 -14952.406} C_VEL
LIN {X 0,Y 326.829,Z 272.043,A -85,B 0,C 180,E1 -14954.952,E2 -14954.952} C_VEL
LIN {X 0,Y 326.387,Z 275.812,A -85,B 0,C 180,E1 -14958.842,E2 -14958.842} C_VEL
LIN {X 0,Y 325.998,Z 279.552,A -85,B 0,C 180,E1 -14962.515,E2 -14962.515} C_VEL
LIN {X 0,Y 327.982,Z 285.532,A -85,B 0,C 180,E1 -14962.978,E2 -14962.978} C_VEL
LIN {X 0,Y 331.447,Z 296.739,A -85,B 0,C 180,E1 -14963.922,E2 -14963.922} C_VEL
LIN {X 0,Y 334.034,Z 308.478,A -85,B 0,C 180,E1 -14965.033,E2 -14965.033} C_VEL
LIN {X 0,Y 334.99,Z 316.554,A -85,B 0,C 180,E1 -14965.863,E2 -14965.863} C_VEL
LIN {X 0,Y 333.627,Z 326.934,A -85,B 0,C 180,E1 -14966.928,E2 -14966.928} C_VEL
LIN {X 0,Y 332.149,Z 337.248,A -85,B 0,C 180,E1 -14968.256,E2 -14968.256} C_VEL
LIN {X 0,Y 330.554,Z 347.434,A -85,B 0,C 180,E1 -14969.881,E2 -14969.881} C_VEL
LIN {X 0,Y 329.309,Z 355.11,A -85,B 0,C 180,E1 -14971.389,E2 -14971.389} C_VEL
LIN {X 0,Y 327.909,Z 362.978,A -85,B 0,C 180,E1 -14973.295,E2 -14973.295} C_VEL
LIN {X 0,Y 326.737,Z 370.068,A -85,B 0,C 180,E1 -14975.502,E2 -14975.502} C_VEL
LIN {X 0,Y 325.792,Z 375.849,A -85,B 0,C 180,E1 -14977.935,E2 -14977.935} C_VEL
LIN {X 0,Y 325.343,Z 378.84,A -85,B 0,C 180,E1 -14979.657,E2 -14979.657} C_VEL
LIN {X 0,Y 324.885,Z 381.653,A -85,B 0,C 180,E1 -14982.111,E2 -14982.111} C_VEL
LIN {X 0,Y 324.656,Z 382.859,A -85,B 0,C 180,E1 -14984.41,E2 -14984.41} C_VEL
LIN {X 0,Y 324.606,Z 382.836,A -85,B 0,C 180,E1 -14986.147,E2 -14986.147} C_VEL
LIN {X 0,Y 324.595,Z 382.058,A -85,B 0,C 180,E1 -14987.842,E2 -14987.842} C_VEL
LIN {X 0,Y 324.741,Z 380.565,A -85,B 0,C 180,E1 -14989.516,E2 -14989.516} C_VEL
LIN {X 0,Y 325.015,Z 378.344,A -85,B 0,C 180,E1 -14991.166,E2 -14991.166} C_VEL
LIN {X 0,Y 325.364,Z 374.823,A -85,B 0,C 180,E1 -14993.052,E2 -14993.052} C_VEL
LIN {X 0,Y 325.871,Z 369.897,A -85,B 0,C 180,E1 -14995.035,E2 -14995.035} C_VEL
LIN {X 0,Y 326.597,Z 363.385,A -85,B 0,C 180,E1 -14997.056,E2 -14997.056} C_VEL
LIN {X 0,Y 327.562,Z 355.438,A -85,B 0,C 180,E1 -14999.008,E2 -14999.008} C_VEL
LIN {X 0,Y 328.605,Z 346.766,A -85,B 0,C 180,E1 -15000.71,E2 -15000.71} C_VEL
LIN {X 0,Y 329.745,Z 336.366,A -85,B 0,C 180,E1 -15002.353,E2 -15002.353} C_VEL
LIN {X 0,Y 330.903,Z 325.884,A -85,B 0,C 180,E1 -15003.682,E2 -15003.682} C_VEL
LIN {X 0,Y 332.009,Z 314.007,A -85,B 0,C 180,E1 -15004.87,E2 -15004.87} C_VEL
LIN {X 0,Y 332.168,Z 311.032,A -85,B 0,C 180,E1 -15005.134,E2 -15005.134} C_VEL
LIN {X 0,Y 330.122,Z 299.224,A -85,B 0,C 180,E1 -15006.141,E2 -15006.141} C_VEL
LIN {X 0,Y 327.393,Z 286.228,A -85,B 0,C 180,E1 -15007.02,E2 -15007.02} C_VEL
LIN {X 0,Y 325.507,Z 278.266,A -85,B 0,C 180,E1 -15007.449,E2 -15007.449} C_VEL
LIN {X 0,Y 325.827,Z 273.471,A -85,B 0,C 180,E1 -15011.628,E2 -15011.628} C_VEL
LIN {X 0,Y 326.055,Z 269.7,A -85,B 0,C 180,E1 -15015.01,E2 -15015.01} C_VEL
LIN {X 0,Y 326.401,Z 265.539,A -85,B 0,C 180,E1 -15018.827,E2 -15018.827} C_VEL
LIN {X 0,Y 326.682,Z 262.791,A -85,B 0,C 180,E1 -15021.503,E2 -15021.503} C_VEL
LIN {X 0,Y 326.922,Z 262.759,A -85,B 0,C 180,E1 -15023.83,E2 -15023.83} C_VEL
LIN {X 0,Y 327.038,Z 262.745,A -85,B 0,C 180,E1 -15027.537,E2 -15027.537} C_VEL
LIN {X 0,Y 327.208,Z 262.725,A -85,B 0,C 180,E1 -15030,E2 -15030} C_VEL
LIN {X 0,Y 327.058,Z 262.748,A -85,B 0,C 180,E1 -15032.463,E2 -15032.463} C_VEL
LIN {X 0,Y 326.986,Z 262.755,A -85,B 0,C 180,E1 -15036.169,E2 -15036.169} C_VEL
LIN {X 0,Y 326.904,Z 262.764,A -85,B 0,C 180,E1 -15038.655,E2 -15038.655} C_VEL
LIN {X 0,Y 326.729,Z 262.787,A -85,B 0,C 180,E1 -15042.421,E2 -15042.421} C_VEL
LIN {X 0,Y 326.744,Z 262.782,A -85,B 0,C 180,E1 -15044.958,E2 -15044.958} C_VEL
LIN {X 0,Y 326.725,Z 262.784,A -85,B 0,C 180,E1 -15048.84,E2 -15048.84} C_VEL
LIN {X 0,Y 326.616,Z 262.797,A -85,B 0,C 180,E1 -15052.787,E2 -15052.787} C_VEL
LIN {X 0,Y 326.681,Z 262.791,A -85,B 0,C 180,E1 -15055.484,E2 -15055.484} C_VEL
LIN {X 0,Y 326.651,Z 262.797,A -85,B 0,C 180,E1 -15059.66,E2 -15059.66} C_VEL
LIN {X 0,Y 326.613,Z 262.798,A -85,B 0,C 180,E1 -15062.948,E2 -15062.948} C_VEL
LIN {X 0,Y 326.623,Z 262.797,A -85,B 0,C 180,E1 -15067.047,E2 -15067.047} C_VEL
LIN {X 0,Y 326.625,Z 262.797,A -85,B 0,C 180,E1 -15070.203,E2 -15070.203} C_VEL
LIN {X 0,Y 326.648,Z 262.798,A -85,B 0,C 180,E1 -15073.51,E2 -15073.51} C_VEL
LIN {X 0,Y 326.64,Z 262.797,A -85,B 0,C 180,E1 -15077.015,E2 -15077.015} C_VEL
LIN {X 0,Y 326.635,Z 262.796,A -85,B 0,C 180,E1 -15080.767,E2 -15080.767} C_VEL
LIN {X 0,Y 326.603,Z 262.799,A -85,B 0,C 180,E1 -15084.481,E2 -15084.481} C_VEL
LIN {X 0,Y 326.599,Z 262.802,A -85,B 0,C 180,E1 -15087.457,E2 -15087.457} C_VEL
LIN {X 0,Y 326.645,Z 262.794,A -85,B 0,C 180,E1 -15090.223,E2 -15090.223} C_VEL
LIN {X 0,Y 326.028,Z 262.875,A -85,B 0,C 180,E1 -15091.252,E2 -15091.252} C_VEL
LIN {X 0,Y 323.195,Z 263.229,A -85,B 0,C 180,E1 -15092.927,E2 -15092.927} C_VEL
LIN {X 0,Y 320.746,Z 263.532,A -85,B 0,C 180,E1 -15094.284,E2 -15094.284} C_VEL
LIN {X 0,Y 319.668,Z 263.665,A -85,B 0,C 180,E1 -15095.335,E2 -15095.335} C_VEL
LIN {X 0,Y 319.568,Z 263.675,A -85,B 0,C 180,E1 -15095.691,E2 -15095.691} C_VEL
LIN {X 0,Y 319.608,Z 263.671,A -85,B 0,C 180,E1 -15099.402,E2 -15099.402} C_VEL
LIN {X 0,Y 319.651,Z 263.666,A -85,B 0,C 180,E1 -15102.074,E2 -15102.074} C_VEL
LIN {X 0,Y 319.725,Z 263.656,A -85,B 0,C 180,E1 -15106.009,E2 -15106.009} C_VEL
LIN {X 0,Y 319.746,Z 263.653,A -85,B 0,C 180,E1 -15109.874,E2 -15109.874} C_VEL
LIN {X 0,Y 319.907,Z 263.638,A -85,B 0,C 180,E1 -15112.427,E2 -15112.427} C_VEL
LIN {X 0,Y 319.74,Z 263.655,A -85,B 0,C 180,E1 -15114.958,E2 -15114.958} C_VEL
LIN {X 0,Y 319.986,Z 263.623,A -85,B 0,C 180,E1 -15117.484,E2 -15117.484} C_VEL
LIN {X 0,Y 320.145,Z 263.607,A -85,B 0,C 180,E1 -15120.001,E2 -15120.001} C_VEL
LIN {X 0,Y 319.987,Z 263.625,A -85,B 0,C 180,E1 -15122.519,E2 -15122.519} C_VEL
LIN {X 0,Y 319.948,Z 263.631,A -85,B 0,C 180,E1 -15126.307,E2 -15126.307} C_VEL
LIN {X 0,Y 319.84,Z 263.641,A -85,B 0,C 180,E1 -15128.849,E2 -15128.849} C_VEL
LIN {X 0,Y 319.681,Z 263.661,A -85,B 0,C 180,E1 -15132.701,E2 -15132.701} C_VEL
LIN {X 0,Y 319.697,Z 263.66,A -85,B 0,C 180,E1 -15135.297,E2 -15135.297} C_VEL
LIN {X 0,Y 319.672,Z 263.663,A -85,B 0,C 180,E1 -15139.257,E2 -15139.257} C_VEL
LIN {X 0,Y 319.569,Z 263.678,A -85,B 0,C 180,E1 -15143.321,E2 -15143.321} C_VEL
LIN {X 0,Y 319.617,Z 263.67,A -85,B 0,C 180,E1 -15146.091,E2 -15146.091} C_VEL
LIN {X 0,Y 319.579,Z 263.675,A -85,B 0,C 180,E1 -15148.936,E2 -15148.936} C_VEL
LIN {X 0,Y 319.53,Z 263.682,A -85,B 0,C 180,E1 -15151.863,E2 -15151.863} C_VEL
LIN {X 0,Y 319.581,Z 263.677,A -85,B 0,C 180,E1 -15155.544,E2 -15155.544} C_VEL
LIN {X 0,Y 319.559,Z 263.677,A -85,B 0,C 180,E1 -15158.011,E2 -15158.011} C_VEL
LIN {X 0,Y 319.527,Z 263.682,A -85,B 0,C 180,E1 -15161.598,E2 -15161.598} C_VEL
LIN {X 0,Y 319.49,Z 263.69,A -85,B 0,C 180,E1 -15165.258,E2 -15165.258} C_VEL
LIN {X 0,Y 319.592,Z 263.835,A -85,B 0,C 180,E1 -15166.66,E2 -15166.66} C_VEL
LIN {X 0,Y 320.409,Z 268.289,A -85,B 0,C 180,E1 -15170.15,E2 -15170.15} C_VEL
LIN {X 0,Y 320.868,Z 272.071,A -85,B 0,C 180,E1 -15172.963,E2 -15172.963} C_VEL
LIN {X 0,Y 320.899,Z 275.345,A -85,B 0,C 180,E1 -15175.29,E2 -15175.29} C_VEL
LIN {X 0,Y 320.18,Z 280.631,A -85,B 0,C 180,E1 -15178.878,E2 -15178.878} C_VEL
LIN {X 0,Y 319.427,Z 287.175,A -85,B 0,C 180,E1 -15183.19,E2 -15183.19} C_VEL
LIN {X 0,Y 318.95,Z 292.517,A -85,B 0,C 180,E1 -15186.633,E2 -15186.633} C_VEL
LIN {X 0,Y 318.8,Z 294.914,A -85,B 0,C 180,E1 -15188.161,E2 -15188.161} C_VEL
LIN {X 0,Y 321.242,Z 308.71,A -85,B 0,C 180,E1 -15188.904,E2 -15188.904} C_VEL
LIN {X 0,Y 323.137,Z 321.273,A -85,B 0,C 180,E1 -15189.811,E2 -15189.811} C_VEL
LIN {X 0,Y 324.382,Z 333.337,A -85,B 0,C 180,E1 -15190.897,E2 -15190.897} C_VEL
LIN {X 0,Y 324.214,Z 337.898,A -85,B 0,C 180,E1 -15191.353,E2 -15191.353} C_VEL
LIN {X 0,Y 322.899,Z 348.789,A -85,B 0,C 180,E1 -15192.586,E2 -15192.586} C_VEL
LIN {X 0,Y 321.788,Z 358.384,A -85,B 0,C 180,E1 -15193.945,E2 -15193.945} C_VEL
LIN {X 0,Y 320.603,Z 368.512,A -85,B 0,C 180,E1 -15195.723,E2 -15195.723} C_VEL
LIN {X 0,Y 319.703,Z 375.827,A -85,B 0,C 180,E1 -15197.301,E2 -15197.301} C_VEL
LIN {X 0,Y 318.88,Z 383.024,A -85,B 0,C 180,E1 -15199.203,E2 -15199.203} C_VEL
LIN {X 0,Y 318.342,Z 388.752,A -85,B 0,C 180,E1 -15201.11,E2 -15201.11} C_VEL
LIN {X 0,Y 317.992,Z 393.249,A -85,B 0,C 180,E1 -15203.018,E2 -15203.018} C_VEL
LIN {X 0,Y 317.819,Z 396.643,A -85,B 0,C 180,E1 -15204.925,E2 -15204.925} C_VEL
LIN {X 0,Y 317.81,Z 398.321,A -85,B 0,C 180,E1 -15206.196,E2 -15206.196} C_VEL
LIN {X 0,Y 317.762,Z 399.584,A -85,B 0,C 180,E1 -15207.465,E2 -15207.465} C_VEL
LIN {X 0,Y 317.747,Z 400.444,A -85,B 0,C 180,E1 -15208.732,E2 -15208.732} C_VEL
LIN {X 0,Y 317.783,Z 400.86,A -85,B 0,C 180,E1 -15210,E2 -15210} C_VEL
LIN {X 0,Y 317.757,Z 400.491,A -85,B 0,C 180,E1 -15212.535,E2 -15212.535} C_VEL
LIN {X 0,Y 317.786,Z 399.721,A -85,B 0,C 180,E1 -15213.804,E2 -15213.804} C_VEL
LIN {X 0,Y 317.829,Z 397.786,A -85,B 0,C 180,E1 -15215.685,E2 -15215.685} C_VEL
LIN {X 0,Y 318.09,Z 394.836,A -85,B 0,C 180,E1 -15217.618,E2 -15217.618} C_VEL
LIN {X 0,Y 318.588,Z 390.893,A -85,B 0,C 180,E1 -15219.523,E2 -15219.523} C_VEL
LIN {X 0,Y 319.343,Z 385.831,A -85,B 0,C 180,E1 -15221.424,E2 -15221.424} C_VEL
LIN {X 0,Y 320.36,Z 379.505,A -85,B 0,C 180,E1 -15223.317,E2 -15223.317} C_VEL
LIN {X 0,Y 321.806,Z 371.635,A -85,B 0,C 180,E1 -15225.192,E2 -15225.192} C_VEL
LIN {X 0,Y 322.902,Z 363.872,A -85,B 0,C 180,E1 -15226.728,E2 -15226.728} C_VEL
LIN {X 0,Y 324.533,Z 354.067,A -85,B 0,C 180,E1 -15228.3,E2 -15228.3} C_VEL
LIN {X 0,Y 326.282,Z 343.462,A -85,B 0,C 180,E1 -15229.667,E2 -15229.667} C_VEL
LIN {X 0,Y 326.988,Z 336.72,A -85,B 0,C 180,E1 -15230.408,E2 -15230.408} C_VEL
LIN {X 0,Y 326.315,Z 326.608,A -85,B 0,C 180,E1 -15231.477,E2 -15231.477} C_VEL
LIN {X 0,Y 324.659,Z 315.167,A -85,B 0,C 180,E1 -15232.537,E2 -15232.537} C_VEL
LIN {X 0,Y 321.846,Z 302.665,A -85,B 0,C 180,E1 -15233.563,E2 -15233.563} C_VEL
LIN {X 0,Y 319.303,Z 293.931,A -85,B 0,C 180,E1 -15234.197,E2 -15234.197} C_VEL
LIN {X 0,Y 319.275,Z 293.573,A -85,B 0,C 180,E1 -15234.25,E2 -15234.25} C_VEL
LIN {X 0,Y 319.994,Z 287.324,A -85,B 0,C 180,E1 -15238.534,E2 -15238.534} C_VEL
LIN {X 0,Y 320.601,Z 282.854,A -85,B 0,C 180,E1 -15241.742,E2 -15241.742} C_VEL
LIN {X 0,Y 321.135,Z 278.963,A -85,B 0,C 180,E1 -15244.68,E2 -15244.68} C_VEL
LIN {X 0,Y 321.306,Z 277.054,A -85,B 0,C 180,E1 -15246.197,E2 -15246.197} C_VEL
LIN {X 0,Y 321.131,Z 273.323,A -85,B 0,C 180,E1 -15249.394,E2 -15249.394} C_VEL
LIN {X 0,Y 320.594,Z 269.756,A -85,B 0,C 180,E1 -15252.809,E2 -15252.809} C_VEL
LIN {X 0,Y 320.033,Z 266.354,A -85,B 0,C 180,E1 -15256.441,E2 -15256.441} C_VEL
LIN {X 0,Y 319.699,Z 264.443,A -85,B 0,C 180,E1 -15258.737,E2 -15258.737} C_VEL
LIN {X 0,Y 319.582,Z 263.681,A -85,B 0,C 180,E1 -15260.375,E2 -15260.375} C_VEL
LIN {X 0,Y 319.558,Z 263.682,A -85,B 0,C 180,E1 -15263.571,E2 -15263.571} C_VEL
LIN {X 0,Y 319.576,Z 263.679,A -85,B 0,C 180,E1 -15266.685,E2 -15266.685} C_VEL
LIN {X 0,Y 319.589,Z 263.677,A -85,B 0,C 180,E1 -15269.615,E2 -15269.615} C_VEL
LIN {X 0,Y 319.606,Z 263.673,A -85,B 0,C 180,E1 -15272.497,E2 -15272.497} C_VEL
LIN {X 0,Y 319.602,Z 263.675,A -85,B 0,C 180,E1 -15275.302,E2 -15275.302} C_VEL
LIN {X 0,Y 319.593,Z 263.677,A -85,B 0,C 180,E1 -15278.046,E2 -15278.046} C_VEL
LIN {X 0,Y 319.685,Z 263.665,A -85,B 0,C 180,E1 -15280.961,E2 -15280.961} C_VEL
LIN {X 0,Y 319.726,Z 263.66,A -85,B 0,C 180,E1 -15285.274,E2 -15285.274} C_VEL
LIN {X 0,Y 319.753,Z 263.657,A -85,B 0,C 180,E1 -15289.871,E2 -15289.871} C_VEL
LIN {X 0,Y 319.927,Z 263.635,A -85,B 0,C 180,E1 -15292.425,E2 -15292.425} C_VEL
LIN {X 0,Y 319.742,Z 263.655,A -85,B 0,C 180,E1 -15294.955,E2 -15294.955} C_VEL
LIN {X 0,Y 319.985,Z 263.629,A -85,B 0,C 180,E1 -15297.481,E2 -15297.481} C_VEL
LIN {X 0,Y 320.143,Z 263.607,A -85,B 0,C 180,E1 -15299.999,E2 -15299.999} C_VEL
LIN {X 0,Y 319.985,Z 263.629,A -85,B 0,C 180,E1 -15302.516,E2 -15302.516} C_VEL
LIN {X 0,Y 319.965,Z 265.032,A -85,B 0,C 180,E1 -15305.039,E2 -15305.039} C_VEL
LIN {X 0,Y 320.295,Z 266.853,A -85,B 0,C 180,E1 -15307.564,E2 -15307.564} C_VEL
LIN {X 0,Y 320.286,Z 268.9,A -85,B 0,C 180,E1 -15310.109,E2 -15310.109} C_VEL
LIN {X 0,Y 319.929,Z 272.258,A -85,B 0,C 180,E1 -15313.982,E2 -15313.982} C_VEL
LIN {X 0,Y 319.447,Z 275.963,A -85,B 0,C 180,E1 -15317.937,E2 -15317.937} C_VEL
LIN {X 0,Y 319.013,Z 279.772,A -85,B 0,C 180,E1 -15321.823,E2 -15321.823} C_VEL
LIN {X 0,Y 321.058,Z 285.792,A -85,B 0,C 180,E1 -15322.316,E2 -15322.316} C_VEL
LIN {X 0,Y 324.79,Z 297.664,A -85,B 0,C 180,E1 -15323.381,E2 -15323.381} C_VEL
LIN {X 0,Y 327.441,Z 309.628,A -85,B 0,C 180,E1 -15324.571,E2 -15324.571} C_VEL
LIN {X 0,Y 328.433,Z 316.711,A -85,B 0,C 180,E1 -15325.337,E2 -15325.337} C_VEL
LIN {X 0,Y 326.987,Z 328.029,A -85,B 0,C 180,E1 -15326.544,E2 -15326.544} C_VEL
LIN {X 0,Y 325.298,Z 339.064,A -85,B 0,C 180,E1 -15328.023,E2 -15328.023} C_VEL
LIN {X 0,Y 323.619,Z 349.015,A -85,B 0,C 180,E1 -15329.697,E2 -15329.697} C_VEL
LIN {X 0,Y 322.083,Z 357.88,A -85,B 0,C 180,E1 -15331.578,E2 -15331.578} C_VEL
LIN {X 0,Y 320.644,Z 365.512,A -85,B 0,C 180,E1 -15333.604,E2 -15333.604} C_VEL
LIN {X 0,Y 319.63,Z 371.262,A -85,B 0,C 180,E1 -15335.557,E2 -15335.557} C_VEL
LIN {X 0,Y 318.857,Z 375.7,A -85,B 0,C 180,E1 -15337.489,E2 -15337.489} C_VEL
LIN {X 0,Y 318.192,Z 379.597,A -85,B 0,C 180,E1 -15339.829,E2 -15339.829} C_VEL
LIN {X 0,Y 317.868,Z 381.524,A -85,B 0,C 180,E1 -15341.549,E2 -15341.549} C_VEL
LIN {X 0,Y 317.647,Z 382.731,A -85,B 0,C 180,E1 -15343.302,E2 -15343.302} C_VEL
LIN {X 0,Y 317.539,Z 383.147,A -85,B 0,C 180,E1 -15345.09,E2 -15345.09} C_VEL
LIN {X 0,Y 317.481,Z 382.746,A -85,B 0,C 180,E1 -15346.927,E2 -15346.927} C_VEL
LIN {X 0,Y 317.574,Z 381.476,A -85,B 0,C 180,E1 -15348.798,E2 -15348.798} C_VEL
LIN {X 0,Y 317.808,Z 379.253,A -85,B 0,C 180,E1 -15350.71,E2 -15350.71} C_VEL
LIN {X 0,Y 318.183,Z 375.944,A -85,B 0,C 180,E1 -15352.668,E2 -15352.668} C_VEL
LIN {X 0,Y 318.685,Z 371.355,A -85,B 0,C 180,E1 -15354.68,E2 -15354.68} C_VEL
LIN {X 0,Y 319.378,Z 365.273,A -85,B 0,C 180,E1 -15356.738,E2 -15356.738} C_VEL
LIN {X 0,Y 320.201,Z 358.51,A -85,B 0,C 180,E1 -15358.552,E2 -15358.552} C_VEL
LIN {X 0,Y 321.265,Z 349.994,A -85,B 0,C 180,E1 -15360.385,E2 -15360.385} C_VEL
LIN {X 0,Y 322.366,Z 340.461,A -85,B 0,C 180,E1 -15362.049,E2 -15362.049} C_VEL
LIN {X 0,Y 323.431,Z 331.507,A -85,B 0,C 180,E1 -15363.322,E2 -15363.322} C_VEL
LIN {X 0,Y 324.622,Z 320.204,A -85,B 0,C 180,E1 -15364.626,E2 -15364.626} C_VEL
LIN {X 0,Y 325.195,Z 311.524,A -85,B 0,C 180,E1 -15365.451,E2 -15365.451} C_VEL
LIN {X 0,Y 323.244,Z 300.142,A -85,B 0,C 180,E1 -15366.453,E2 -15366.453} C_VEL
LIN {X 0,Y 320.43,Z 286.77,A -85,B 0,C 180,E1 -15367.387,E2 -15367.387} C_VEL
LIN {X 0,Y 318.485,Z 278.411,A -85,B 0,C 180,E1 -15367.891,E2 -15367.891} C_VEL
LIN {X 0,Y 318.798,Z 273.766,A -85,B 0,C 180,E1 -15372.024,E2 -15372.024} C_VEL
LIN {X 0,Y 319.112,Z 269.437,A -85,B 0,C 180,E1 -15375.981,E2 -15375.981} C_VEL
LIN {X 0,Y 319.441,Z 265.313,A -85,B 0,C 180,E1 -15379.863,E2 -15379.863} C_VEL
LIN {X 0,Y 319.674,Z 263.664,A -85,B 0,C 180,E1 -15381.605,E2 -15381.605} C_VEL
LIN {X 0,Y 319.872,Z 263.637,A -85,B 0,C 180,E1 -15383.693,E2 -15383.693} C_VEL
LIN {X 0,Y 319.981,Z 263.624,A -85,B 0,C 180,E1 -15387.483,E2 -15387.483} C_VEL
LIN {X 0,Y 320.159,Z 263.603,A -85,B 0,C 180,E1 -15390,E2 -15390} C_VEL
LIN {X 0,Y 319.999,Z 263.627,A -85,B 0,C 180,E1 -15392.518,E2 -15392.518} C_VEL
LIN {X 0,Y 319.942,Z 263.633,A -85,B 0,C 180,E1 -15396.306,E2 -15396.306} C_VEL
LIN {X 0,Y 319.833,Z 263.644,A -85,B 0,C 180,E1 -15398.848,E2 -15398.848} C_VEL
LIN {X 0,Y 319.675,Z 263.664,A -85,B 0,C 180,E1 -15402.7,E2 -15402.7} C_VEL
LIN {X 0,Y 319.69,Z 263.66,A -85,B 0,C 180,E1 -15405.296,E2 -15405.296} C_VEL
LIN {X 0,Y 319.667,Z 263.663,A -85,B 0,C 180,E1 -15409.255,E2 -15409.255} C_VEL
LIN {X 0,Y 319.566,Z 263.676,A -85,B 0,C 180,E1 -15413.319,E2 -15413.319} C_VEL
LIN {X 0,Y 319.626,Z 263.671,A -85,B 0,C 180,E1 -15416.089,E2 -15416.089} C_VEL
LIN {X 0,Y 319.58,Z 263.673,A -85,B 0,C 180,E1 -15418.934,E2 -15418.934} C_VEL
LIN {X 0,Y 319.528,Z 263.685,A -85,B 0,C 180,E1 -15421.862,E2 -15421.862} C_VEL
LIN {X 0,Y 319.571,Z 263.68,A -85,B 0,C 180,E1 -15425.544,E2 -15425.544} C_VEL
LIN {X 0,Y 319.59,Z 263.674,A -85,B 0,C 180,E1 -15428.005,E2 -15428.005} C_VEL
LIN {X 0,Y 319.592,Z 263.676,A -85,B 0,C 180,E1 -15431.613,E2 -15431.613} C_VEL
LIN {X 0,Y 319.636,Z 263.671,A -85,B 0,C 180,E1 -15435.286,E2 -15435.286} C_VEL
LIN {X 0,Y 319.573,Z 263.676,A -85,B 0,C 180,E1 -15438.721,E2 -15438.721} C_VEL
LIN {X 0,Y 319.573,Z 263.675,A -85,B 0,C 180,E1 -15442.344,E2 -15442.344} C_VEL
LIN {X 0,Y 319.551,Z 263.683,A -85,B 0,C 180,E1 -15445.125,E2 -15445.125} C_VEL
LIN {X 0,Y 319.562,Z 263.68,A -85,B 0,C 180,E1 -15449.059,E2 -15449.059} C_VEL
LIN {X 0,Y 319.601,Z 263.672,A -85,B 0,C 180,E1 -15452.499,E2 -15452.499} C_VEL
LIN {X 0,Y 319.568,Z 263.675,A -85,B 0,C 180,E1 -15455.691,E2 -15455.691} C_VEL
LIN {X 0,Y 318.877,Z 263.766,A -85,B 0,C 180,E1 -15456.743,E2 -15456.743} C_VEL
LIN {X 0,Y 316.053,Z 264.117,A -85,B 0,C 180,E1 -15458.456,E2 -15458.456} C_VEL
LIN {X 0,Y 313.69,Z 264.412,A -85,B 0,C 180,E1 -15459.844,E2 -15459.844} C_VEL
LIN {X 0,Y 312.693,Z 264.535,A -85,B 0,C 180,E1 -15460.918,E2 -15460.918} C_VEL
LIN {X 0,Y 312.618,Z 264.542,A -85,B 0,C 180,E1 -15461.281,E2 -15461.281} C_VEL
LIN {X 0,Y 312.687,Z 264.531,A -85,B 0,C 180,E1 -15465.688,E2 -15465.688} C_VEL
LIN {X 0,Y 312.692,Z 264.53,A -85,B 0,C 180,E1 -15469.643,E2 -15469.643} C_VEL
LIN {X 0,Y 312.847,Z 264.515,A -85,B 0,C 180,E1 -15472.255,E2 -15472.255} C_VEL
LIN {X 0,Y 312.71,Z 264.531,A -85,B 0,C 180,E1 -15474.844,E2 -15474.844} C_VEL
LIN {X 0,Y 312.985,Z 264.497,A -85,B 0,C 180,E1 -15478.715,E2 -15478.715} C_VEL
LIN {X 0,Y 312.986,Z 264.495,A -85,B 0,C 180,E1 -15481.288,E2 -15481.288} C_VEL
LIN {X 0,Y 312.714,Z 264.527,A -85,B 0,C 180,E1 -15485.159,E2 -15485.159} C_VEL
LIN {X 0,Y 312.868,Z 264.512,A -85,B 0,C 180,E1 -15487.747,E2 -15487.747} C_VEL
LIN {X 0,Y 312.669,Z 264.538,A -85,B 0,C 180,E1 -15491.673,E2 -15491.673} C_VEL
LIN {X 0,Y 312.698,Z 264.531,A -85,B 0,C 180,E1 -15494.889,E2 -15494.889} C_VEL
LIN {X 0,Y 312.628,Z 264.54,A -85,B 0,C 180,E1 -15499.238,E2 -15499.238} C_VEL
LIN {X 0,Y 312.545,Z 264.55,A -85,B 0,C 180,E1 -15502.791,E2 -15502.791} C_VEL
LIN {X 0,Y 312.596,Z 264.546,A -85,B 0,C 180,E1 -15505.935,E2 -15505.935} C_VEL
LIN {X 0,Y 312.538,Z 264.555,A -85,B 0,C 180,E1 -15509.652,E2 -15509.652} C_VEL
LIN {X 0,Y 312.52,Z 264.556,A -85,B 0,C 180,E1 -15513.69,E2 -15513.69} C_VEL
LIN {X 0,Y 312.527,Z 264.557,A -85,B 0,C 180,E1 -15517.386,E2 -15517.386} C_VEL
LIN {X 0,Y 312.491,Z 264.558,A -85,B 0,C 180,E1 -15520.71,E2 -15520.71} C_VEL
LIN {X 0,Y 312.453,Z 264.562,A -85,B 0,C 180,E1 -15524.211,E2 -15524.211} C_VEL
LIN {X 0,Y 312.565,Z 264.764,A -85,B 0,C 180,E1 -15526.482,E2 -15526.482} C_VEL
LIN {X 0,Y 313.276,Z 268.783,A -85,B 0,C 180,E1 -15529.709,E2 -15529.709} C_VEL
LIN {X 0,Y 313.812,Z 272.822,A -85,B 0,C 180,E1 -15532.795,E2 -15532.795} C_VEL
LIN {X 0,Y 313.881,Z 276.104,A -85,B 0,C 180,E1 -15535.183,E2 -15535.183} C_VEL
LIN {X 0,Y 313.108,Z 281.487,A -85,B 0,C 180,E1 -15538.919,E2 -15538.919} C_VEL
LIN {X 0,Y 312.336,Z 287.915,A -85,B 0,C 180,E1 -15543.255,E2 -15543.255} C_VEL
LIN {X 0,Y 311.775,Z 294.654,A -85,B 0,C 180,E1 -15547.69,E2 -15547.69} C_VEL
LIN {X 0,Y 311.868,Z 295.621,A -85,B 0,C 180,E1 -15547.785,E2 -15547.785} C_VEL
LIN {X 0,Y 314.278,Z 308.882,A -85,B 0,C 180,E1 -15548.533,E2 -15548.533} C_VEL
LIN {X 0,Y 316.236,Z 322.174,A -85,B 0,C 180,E1 -15549.531,E2 -15549.531} C_VEL
LIN {X 0,Y 317.405,Z 333.62,A -85,B 0,C 180,E1 -15550.602,E2 -15550.602} C_VEL
LIN {X 0,Y 317.283,Z 338.397,A -85,B 0,C 180,E1 -15551.098,E2 -15551.098} C_VEL
LIN {X 0,Y 315.926,Z 349.114,A -85,B 0,C 180,E1 -15552.356,E2 -15552.356} C_VEL
LIN {X 0,Y 314.803,Z 358.58,A -85,B 0,C 180,E1 -15553.739,E2 -15553.739} C_VEL
LIN {X 0,Y 313.673,Z 367.86,A -85,B 0,C 180,E1 -15555.401,E2 -15555.401} C_VEL
LIN {X 0,Y 312.734,Z 375.251,A -85,B 0,C 180,E1 -15557.013,E2 -15557.013} C_VEL
LIN {X 0,Y 311.841,Z 382.524,A -85,B 0,C 180,E1 -15558.956,E2 -15558.956} C_VEL
LIN {X 0,Y 311.281,Z 388.327,A -85,B 0,C 180,E1 -15560.907,E2 -15560.907} C_VEL
LIN {X 0,Y 310.922,Z 392.878,A -85,B 0,C 180,E1 -15562.858,E2 -15562.858} C_VEL
LIN {X 0,Y 310.727,Z 396.318,A -85,B 0,C 180,E1 -15564.809,E2 -15564.809} C_VEL
LIN {X 0,Y 310.721,Z 398.02,A -85,B 0,C 180,E1 -15566.109,E2 -15566.109} C_VEL
LIN {X 0,Y 310.685,Z 399.307,A -85,B 0,C 180,E1 -15567.407,E2 -15567.407} C_VEL
LIN {X 0,Y 310.661,Z 400.191,A -85,B 0,C 180,E1 -15568.704,E2 -15568.704} C_VEL
LIN {X 0,Y 310.693,Z 400.647,A -85,B 0,C 180,E1 -15570,E2 -15570} C_VEL
LIN {X 0,Y 310.679,Z 400.319,A -85,B 0,C 180,E1 -15572.593,E2 -15572.593} C_VEL
LIN {X 0,Y 310.699,Z 399.57,A -85,B 0,C 180,E1 -15573.891,E2 -15573.891} C_VEL
LIN {X 0,Y 310.728,Z 397.907,A -85,B 0,C 180,E1 -15575.615,E2 -15575.615} C_VEL
LIN {X 0,Y 311.033,Z 394.766,A -85,B 0,C 180,E1 -15577.791,E2 -15577.791} C_VEL
LIN {X 0,Y 311.552,Z 390.866,A -85,B 0,C 180,E1 -15579.74,E2 -15579.74} C_VEL
LIN {X 0,Y 312.339,Z 385.867,A -85,B 0,C 180,E1 -15581.683,E2 -15581.683} C_VEL
LIN {X 0,Y 313.46,Z 379.617,A -85,B 0,C 180,E1 -15583.616,E2 -15583.616} C_VEL
LIN {X 0,Y 314.957,Z 371.866,A -85,B 0,C 180,E1 -15585.531,E2 -15585.531} C_VEL
LIN {X 0,Y 316.239,Z 363.434,A -85,B 0,C 180,E1 -15587.233,E2 -15587.233} C_VEL
LIN {X 0,Y 318.004,Z 353.427,A -85,B 0,C 180,E1 -15588.857,E2 -15588.857} C_VEL
LIN {X 0,Y 319.846,Z 342.722,A -85,B 0,C 180,E1 -15590.247,E2 -15590.247} C_VEL
LIN {X 0,Y 320.338,Z 337.439,A -85,B 0,C 180,E1 -15590.85,E2 -15590.85} C_VEL
LIN {X 0,Y 319.581,Z 326.315,A -85,B 0,C 180,E1 -15592.073,E2 -15592.073} C_VEL
LIN {X 0,Y 317.829,Z 314.554,A -85,B 0,C 180,E1 -15593.209,E2 -15593.209} C_VEL
LIN {X 0,Y 315.149,Z 303.021,A -85,B 0,C 180,E1 -15594.199,E2 -15594.199} C_VEL
LIN {X 0,Y 312.329,Z 293.704,A -85,B 0,C 180,E1 -15594.919,E2 -15594.919} C_VEL
LIN {X 0,Y 312.3,Z 293.283,A -85,B 0,C 180,E1 -15595.02,E2 -15595.02} C_VEL
LIN {X 0,Y 313.031,Z 287.817,A -85,B 0,C 180,E1 -15598.881,E2 -15598.881} C_VEL
LIN {X 0,Y 313.736,Z 282.911,A -85,B 0,C 180,E1 -15602.521,E2 -15602.521} C_VEL
LIN {X 0,Y 314.227,Z 279.063,A -85,B 0,C 180,E1 -15605.556,E2 -15605.556} C_VEL
LIN {X 0,Y 314.231,Z 275.65,A -85,B 0,C 180,E1 -15608.481,E2 -15608.481} C_VEL
LIN {X 0,Y 314.005,Z 273.495,A -85,B 0,C 180,E1 -15610.471,E2 -15610.471} C_VEL
LIN {X 0,Y 313.424,Z 269.889,A -85,B 0,C 180,E1 -15614.146,E2 -15614.146} C_VEL
LIN {X 0,Y 312.913,Z 266.704,A -85,B 0,C 180,E1 -15617.83,E2 -15617.83} C_VEL
LIN {X 0,Y 312.531,Z 264.559,A -85,B 0,C 180,E1 -15620.974,E2 -15620.974} C_VEL
LIN {X 0,Y 312.531,Z 264.556,A -85,B 0,C 180,E1 -15624.219,E2 -15624.219} C_VEL
LIN {X 0,Y 312.503,Z 264.559,A -85,B 0,C 180,E1 -15627.332,E2 -15627.332} C_VEL
LIN {X 0,Y 312.55,Z 264.552,A -85,B 0,C 180,E1 -15631.275,E2 -15631.275} C_VEL
LIN {X 0,Y 312.583,Z 264.549,A -85,B 0,C 180,E1 -15634.709,E2 -15634.709} C_VEL
LIN {X 0,Y 312.584,Z 264.549,A -85,B 0,C 180,E1 -15637.527,E2 -15637.527} C_VEL
LIN {X 0,Y 312.634,Z 264.543,A -85,B 0,C 180,E1 -15641.655,E2 -15641.655} C_VEL
LIN {X 0,Y 312.689,Z 264.537,A -85,B 0,C 180,E1 -15645.685,E2 -15645.685} C_VEL
LIN {X 0,Y 312.697,Z 264.536,A -85,B 0,C 180,E1 -15649.64,E2 -15649.64} C_VEL
LIN {X 0,Y 312.866,Z 264.514,A -85,B 0,C 180,E1 -15652.253,E2 -15652.253} C_VEL
LIN {X 0,Y 312.712,Z 264.531,A -85,B 0,C 180,E1 -15654.841,E2 -15654.841} C_VEL
LIN {X 0,Y 312.984,Z 264.499,A -85,B 0,C 180,E1 -15658.712,E2 -15658.712} C_VEL
LIN {X 0,Y 312.984,Z 264.5,A -85,B 0,C 180,E1 -15661.285,E2 -15661.285} C_VEL
LIN {X 0,Y 312.964,Z 264.701,A -85,B 0,C 180,E1 -15662.573,E2 -15662.573} C_VEL
LIN {X 0,Y 313.217,Z 267.608,A -85,B 0,C 180,E1 -15666.82,E2 -15666.82} C_VEL
LIN {X 0,Y 313.336,Z 269.46,A -85,B 0,C 180,E1 -15669.291,E2 -15669.291} C_VEL
LIN {X 0,Y 312.998,Z 272.528,A -85,B 0,C 180,E1 -15672.974,E2 -15672.974} C_VEL
LIN {X 0,Y 312.694,Z 274.894,A -85,B 0,C 180,E1 -15675.645,E2 -15675.645} C_VEL
LIN {X 0,Y 312.298,Z 278.069,A -85,B 0,C 180,E1 -15679.064,E2 -15679.064} C_VEL
LIN {X 0,Y 312.058,Z 280.056,A -85,B 0,C 180,E1 -15681.119,E2 -15681.119} C_VEL
LIN {X 0,Y 313.963,Z 285.721,A -85,B 0,C 180,E1 -15681.587,E2 -15681.587} C_VEL
LIN {X 0,Y 317.608,Z 296.538,A -85,B 0,C 180,E1 -15682.602,E2 -15682.602} C_VEL
LIN {X 0,Y 320.44,Z 308.555,A -85,B 0,C 180,E1 -15683.833,E2 -15683.833} C_VEL
LIN {X 0,Y 321.843,Z 317.554,A -85,B 0,C 180,E1 -15684.855,E2 -15684.855} C_VEL
LIN {X 0,Y 320.279,Z 329.625,A -85,B 0,C 180,E1 -15686.205,E2 -15686.205} C_VEL
LIN {X 0,Y 318.67,Z 339.597,A -85,B 0,C 180,E1 -15687.588,E2 -15687.588} C_VEL
LIN {X 0,Y 316.989,Z 348.964,A -85,B 0,C 180,E1 -15689.192,E2 -15689.192} C_VEL
LIN {X 0,Y 315.372,Z 357.782,A -85,B 0,C 180,E1 -15691.087,E2 -15691.087} C_VEL
LIN {X 0,Y 313.801,Z 365.594,A -85,B 0,C 180,E1 -15693.19,E2 -15693.19} C_VEL
LIN {X 0,Y 312.628,Z 371.814,A -85,B 0,C 180,E1 -15695.369,E2 -15695.369} C_VEL
LIN {X 0,Y 311.771,Z 376.436,A -85,B 0,C 180,E1 -15697.489,E2 -15697.489} C_VEL
LIN {X 0,Y 311.111,Z 380.099,A -85,B 0,C 180,E1 -15699.822,E2 -15699.822} C_VEL
LIN {X 0,Y 310.748,Z 382.038,A -85,B 0,C 180,E1 -15701.727,E2 -15701.727} C_VEL
LIN {X 0,Y 310.516,Z 383.089,A -85,B 0,C 180,E1 -15703.594,E2 -15703.594} C_VEL
LIN {X 0,Y 310.422,Z 383.328,A -85,B 0,C 180,E1 -15705.426,E2 -15705.426} C_VEL
LIN {X 0,Y 310.395,Z 382.804,A -85,B 0,C 180,E1 -15707.215,E2 -15707.215} C_VEL
LIN {X 0,Y 310.486,Z 381.501,A -85,B 0,C 180,E1 -15708.973,E2 -15708.973} C_VEL
LIN {X 0,Y 310.724,Z 379.487,A -85,B 0,C 180,E1 -15710.707,E2 -15710.707} C_VEL
LIN {X 0,Y 311.034,Z 376.777,A -85,B 0,C 180,E1 -15712.406,E2 -15712.406} C_VEL
LIN {X 0,Y 311.496,Z 372.754,A -85,B 0,C 180,E1 -15714.311,E2 -15714.311} C_VEL
LIN {X 0,Y 312.134,Z 366.976,A -85,B 0,C 180,E1 -15716.414,E2 -15716.414} C_VEL
LIN {X 0,Y 313.069,Z 359.509,A -85,B 0,C 180,E1 -15718.541,E2 -15718.541} C_VEL
LIN {X 0,Y 314.24,Z 350.657,A -85,B 0,C 180,E1 -15720.527,E2 -15720.527} C_VEL
LIN {X 0,Y 315.436,Z 340.716,A -85,B 0,C 180,E1 -15722.308,E2 -15722.308} C_VEL
LIN {X 0,Y 316.694,Z 330.132,A -85,B 0,C 180,E1 -15723.825,E2 -15723.825} C_VEL
LIN {X 0,Y 317.972,Z 318.227,A -85,B 0,C 180,E1 -15725.169,E2 -15725.169} C_VEL
LIN {X 0,Y 318.286,Z 312.539,A -85,B 0,C 180,E1 -15725.717,E2 -15725.717} C_VEL
LIN {X 0,Y 316.373,Z 300.98,A -85,B 0,C 180,E1 -15726.778,E2 -15726.778} C_VEL
LIN {X 0,Y 313.539,Z 287.64,A -85,B 0,C 180,E1 -15727.751,E2 -15727.751} C_VEL
LIN {X 0,Y 311.415,Z 278.625,A -85,B 0,C 180,E1 -15728.277,E2 -15728.277} C_VEL
LIN {X 0,Y 311.688,Z 274.964,A -85,B 0,C 180,E1 -15731.599,E2 -15731.599} C_VEL
LIN {X 0,Y 312.049,Z 270.598,A -85,B 0,C 180,E1 -15735.656,E2 -15735.656} C_VEL
LIN {X 0,Y 312.355,Z 266.439,A -85,B 0,C 180,E1 -15739.631,E2 -15739.631} C_VEL
LIN {X 0,Y 312.604,Z 264.545,A -85,B 0,C 180,E1 -15741.562,E2 -15741.562} C_VEL
LIN {X 0,Y 312.806,Z 264.518,A -85,B 0,C 180,E1 -15743.55,E2 -15743.55} C_VEL
LIN {X 0,Y 312.928,Z 264.503,A -85,B 0,C 180,E1 -15747.426,E2 -15747.426} C_VEL
LIN {X 0,Y 313.111,Z 264.481,A -85,B 0,C 180,E1 -15750,E2 -15750} C_VEL
LIN {X 0,Y 312.942,Z 264.505,A -85,B 0,C 180,E1 -15752.574,E2 -15752.574} C_VEL
LIN {X 0,Y 312.9,Z 264.511,A -85,B 0,C 180,E1 -15756.448,E2 -15756.448} C_VEL
LIN {X 0,Y 312.778,Z 264.522,A -85,B 0,C 180,E1 -15759.049,E2 -15759.049} C_VEL
LIN {X 0,Y 312.627,Z 264.54,A -85,B 0,C 180,E1 -15762.991,E2 -15762.991} C_VEL
LIN {X 0,Y 312.628,Z 264.541,A -85,B 0,C 180,E1 -15765.65,E2 -15765.65} C_VEL
LIN {X 0,Y 312.597,Z 264.546,A -85,B 0,C 180,E1 -15769.709,E2 -15769.709} C_VEL
LIN {X 0,Y 312.539,Z 264.551,A -85,B 0,C 180,E1 -15772.791,E2 -15772.791} C_VEL
LIN {X 0,Y 312.594,Z 264.548,A -85,B 0,C 180,E1 -15775.937,E2 -15775.937} C_VEL
LIN {X 0,Y 312.536,Z 264.554,A -85,B 0,C 180,E1 -15779.65,E2 -15779.65} C_VEL
LIN {X 0,Y 312.51,Z 264.56,A -85,B 0,C 180,E1 -15783.69,E2 -15783.69} C_VEL
LIN {X 0,Y 312.543,Z 264.554,A -85,B 0,C 180,E1 -15787.382,E2 -15787.382} C_VEL
LIN {X 0,Y 312.525,Z 264.551,A -85,B 0,C 180,E1 -15790.703,E2 -15790.703} C_VEL
LIN {X 0,Y 312.585,Z 264.544,A -85,B 0,C 180,E1 -15794.185,E2 -15794.185} C_VEL
LIN {X 0,Y 312.547,Z 264.551,A -85,B 0,C 180,E1 -15797.905,E2 -15797.905} C_VEL
LIN {X 0,Y 312.536,Z 264.552,A -85,B 0,C 180,E1 -15801.909,E2 -15801.909} C_VEL
LIN {X 0,Y 312.497,Z 264.556,A -85,B 0,C 180,E1 -15805.791,E2 -15805.791} C_VEL
LIN {X 0,Y 312.515,Z 264.556,A -85,B 0,C 180,E1 -15808.855,E2 -15808.855} C_VEL
LIN {X 0,Y 312.566,Z 264.546,A -85,B 0,C 180,E1 -15811.826,E2 -15811.826} C_VEL
LIN {X 0,Y 312.577,Z 264.549,A -85,B 0,C 180,E1 -15814.712,E2 -15814.712} C_VEL
LIN {X 0,Y 312.58,Z 264.546,A -85,B 0,C 180,E1 -15817.53,E2 -15817.53} C_VEL
LIN {X 0,Y 312.618,Z 264.542,A -85,B 0,C 180,E1 -15821.281,E2 -15821.281} C_VEL
LIN {X 0,Y 311.972,Z 264.625,A -85,B 0,C 180,E1 -15822.358,E2 -15822.358} C_VEL
LIN {X 0,Y 309.134,Z 264.977,A -85,B 0,C 180,E1 -15824.111,E2 -15824.111} C_VEL
LIN {X 0,Y 306.71,Z 265.28,A -85,B 0,C 180,E1 -15825.532,E2 -15825.532} C_VEL
LIN {X 0,Y 305.66,Z 265.409,A -85,B 0,C 180,E1 -15826.632,E2 -15826.632} C_VEL
LIN {X 0,Y 305.571,Z 265.417,A -85,B 0,C 180,E1 -15827.005,E2 -15827.005} C_VEL
LIN {X 0,Y 305.768,Z 265.393,A -85,B 0,C 180,E1 -15831.237,E2 -15831.237} C_VEL
LIN {X 0,Y 305.837,Z 265.385,A -85,B 0,C 180,E1 -15833.404,E2 -15833.404} C_VEL
LIN {X 0,Y 305.881,Z 265.38,A -85,B 0,C 180,E1 -15837.368,E2 -15837.368} C_VEL
LIN {X 0,Y 306.05,Z 265.362,A -85,B 0,C 180,E1 -15840.002,E2 -15840.002} C_VEL
LIN {X 0,Y 305.882,Z 265.38,A -85,B 0,C 180,E1 -15842.635,E2 -15842.635} C_VEL
LIN {X 0,Y 305.848,Z 265.384,A -85,B 0,C 180,E1 -15846.599,E2 -15846.599} C_VEL
LIN {X 0,Y 305.733,Z 265.398,A -85,B 0,C 180,E1 -15849.261,E2 -15849.261} C_VEL
LIN {X 0,Y 305.588,Z 265.418,A -85,B 0,C 180,E1 -15853.298,E2 -15853.298} C_VEL
LIN {X 0,Y 305.592,Z 265.419,A -85,B 0,C 180,E1 -15856.022,E2 -15856.022} C_VEL
LIN {X 0,Y 305.575,Z 265.419,A -85,B 0,C 180,E1 -15859.446,E2 -15859.446} C_VEL
LIN {X 0,Y 305.489,Z 265.43,A -85,B 0,C 180,E1 -15863.043,E2 -15863.043} C_VEL
LIN {X 0,Y 305.525,Z 265.425,A -85,B 0,C 180,E1 -15866.22,E2 -15866.22} C_VEL
LIN {X 0,Y 305.487,Z 265.43,A -85,B 0,C 180,E1 -15869.049,E2 -15869.049} C_VEL
LIN {X 0,Y 305.442,Z 265.437,A -85,B 0,C 180,E1 -15871.954,E2 -15871.954} C_VEL
LIN {X 0,Y 305.463,Z 265.436,A -85,B 0,C 180,E1 -15875.115,E2 -15875.115} C_VEL
LIN {X 0,Y 305.451,Z 265.435,A -85,B 0,C 180,E1 -15878.53,E2 -15878.53} C_VEL
LIN {X 0,Y 305.456,Z 265.435,A -85,B 0,C 180,E1 -15882.587,E2 -15882.587} C_VEL
LIN {X 0,Y 305.479,Z 265.631,A -85,B 0,C 180,E1 -15886.243,E2 -15886.243} C_VEL
LIN {X 0,Y 306.334,Z 270.247,A -85,B 0,C 180,E1 -15890.031,E2 -15890.031} C_VEL
LIN {X 0,Y 306.69,Z 272.469,A -85,B 0,C 180,E1 -15891.778,E2 -15891.778} C_VEL
LIN {X 0,Y 306.831,Z 276.844,A -85,B 0,C 180,E1 -15895.067,E2 -15895.067} C_VEL
LIN {X 0,Y 306.039,Z 282.233,A -85,B 0,C 180,E1 -15898.889,E2 -15898.889} C_VEL
LIN {X 0,Y 305.327,Z 287.585,A -85,B 0,C 180,E1 -15902.59,E2 -15902.59} C_VEL
LIN {X 0,Y 304.844,Z 292.915,A -85,B 0,C 180,E1 -15906.206,E2 -15906.206} C_VEL
LIN {X 0,Y 304.715,Z 294.556,A -85,B 0,C 180,E1 -15907.307,E2 -15907.307} C_VEL
LIN {X 0,Y 307.218,Z 308.066,A -85,B 0,C 180,E1 -15908.079,E2 -15908.079} C_VEL
LIN {X 0,Y 309.159,Z 321.688,A -85,B 0,C 180,E1 -15909.119,E2 -15909.119} C_VEL
LIN {X 0,Y 310.305,Z 332.394,A -85,B 0,C 180,E1 -15910.14,E2 -15910.14} C_VEL
LIN {X 0,Y 310.532,Z 337.328,A -85,B 0,C 180,E1 -15910.671,E2 -15910.671} C_VEL
LIN {X 0,Y 309.13,Z 348.252,A -85,B 0,C 180,E1 -15911.955,E2 -15911.955} C_VEL
LIN {X 0,Y 307.802,Z 358.85,A -85,B 0,C 180,E1 -15913.536,E2 -15913.536} C_VEL
LIN {X 0,Y 306.542,Z 368.837,A -85,B 0,C 180,E1 -15915.393,E2 -15915.393} C_VEL
LIN {X 0,Y 305.413,Z 377.297,A -85,B 0,C 180,E1 -15917.373,E2 -15917.373} C_VEL
LIN {X 0,Y 304.63,Z 384.103,A -85,B 0,C 180,E1 -15919.364,E2 -15919.364} C_VEL
LIN {X 0,Y 304.1,Z 389.534,A -85,B 0,C 180,E1 -15921.36,E2 -15921.36} C_VEL
LIN {X 0,Y 303.753,Z 393.756,A -85,B 0,C 180,E1 -15923.357,E2 -15923.357} C_VEL
LIN {X 0,Y 303.642,Z 395.985,A -85,B 0,C 180,E1 -15924.688,E2 -15924.688} C_VEL
LIN {X 0,Y 303.635,Z 397.72,A -85,B 0,C 180,E1 -15926.018,E2 -15926.018} C_VEL
LIN {X 0,Y 303.61,Z 399.029,A -85,B 0,C 180,E1 -15927.346,E2 -15927.346} C_VEL
LIN {X 0,Y 303.578,Z 399.935,A -85,B 0,C 180,E1 -15928.673,E2 -15928.673} C_VEL
LIN {X 0,Y 303.606,Z 400.432,A -85,B 0,C 180,E1 -15930,E2 -15930} C_VEL
LIN {X 0,Y 303.567,Z 400.485,A -85,B 0,C 180,E1 -15931.326,E2 -15931.326} C_VEL
LIN {X 0,Y 303.604,Z 400.147,A -85,B 0,C 180,E1 -15932.653,E2 -15932.653} C_VEL
LIN {X 0,Y 303.594,Z 399.418,A -85,B 0,C 180,E1 -15933.982,E2 -15933.982} C_VEL
LIN {X 0,Y 303.63,Z 398.028,A -85,B 0,C 180,E1 -15935.544,E2 -15935.544} C_VEL
LIN {X 0,Y 303.997,Z 394.713,A -85,B 0,C 180,E1 -15937.973,E2 -15937.973} C_VEL
LIN {X 0,Y 304.524,Z 390.875,A -85,B 0,C 180,E1 -15939.967,E2 -15939.967} C_VEL
LIN {X 0,Y 305.348,Z 385.932,A -85,B 0,C 180,E1 -15941.955,E2 -15941.955} C_VEL
LIN {X 0,Y 306.571,Z 379.742,A -85,B 0,C 180,E1 -15943.928,E2 -15943.928} C_VEL
LIN {X 0,Y 308.119,Z 372.089,A -85,B 0,C 180,E1 -15945.885,E2 -15945.885} C_VEL
LIN {X 0,Y 309.34,Z 364.494,A -85,B 0,C 180,E1 -15947.485,E2 -15947.485} C_VEL
LIN {X 0,Y 311.13,Z 354.919,A -85,B 0,C 180,E1 -15949.119,E2 -15949.119} C_VEL
LIN {X 0,Y 313.032,Z 344.611,A -85,B 0,C 180,E1 -15950.536,E2 -15950.536} C_VEL
LIN {X 0,Y 313.711,Z 339.44,A -85,B 0,C 180,E1 -15951.157,E2 -15951.157} C_VEL
LIN {X 0,Y 313.15,Z 328.635,A -85,B 0,C 180,E1 -15952.428,E2 -15952.428} C_VEL
LIN {X 0,Y 311.633,Z 317.323,A -85,B 0,C 180,E1 -15953.599,E2 -15953.599} C_VEL
LIN {X 0,Y 308.999,Z 305.44,A -85,B 0,C 180,E1 -15954.698,E2 -15954.698} C_VEL
LIN {X 0,Y 305.437,Z 293.688,A -85,B 0,C 180,E1 -15955.688,E2 -15955.688} C_VEL
LIN {X 0,Y 305.374,Z 293.143,A -85,B 0,C 180,E1 -15955.732,E2 -15955.732} C_VEL
LIN {X 0,Y 306.047,Z 288.342,A -85,B 0,C 180,E1 -15959.233,E2 -15959.233} C_VEL
LIN {X 0,Y 306.862,Z 282.993,A -85,B 0,C 180,E1 -15963.343,E2 -15963.343} C_VEL
LIN {X 0,Y 307.313,Z 279.183,A -85,B 0,C 180,E1 -15966.483,E2 -15966.483} C_VEL
LIN {X 0,Y 307.206,Z 276.461,A -85,B 0,C 180,E1 -15968.937,E2 -15968.937} C_VEL
LIN {X 0,Y 306.835,Z 273.722,A -85,B 0,C 180,E1 -15971.623,E2 -15971.623} C_VEL
LIN {X 0,Y 306.293,Z 270.288,A -85,B 0,C 180,E1 -15975.34,E2 -15975.34} C_VEL
LIN {X 0,Y 305.746,Z 267.084,A -85,B 0,C 180,E1 -15979.335,E2 -15979.335} C_VEL
LIN {X 0,Y 305.508,Z 265.492,A -85,B 0,C 180,E1 -15981.601,E2 -15981.601} C_VEL
LIN {X 0,Y 305.461,Z 265.437,A -85,B 0,C 180,E1 -15984.885,E2 -15984.885} C_VEL
LIN {X 0,Y 305.45,Z 265.438,A -85,B 0,C 180,E1 -15988.353,E2 -15988.353} C_VEL
LIN {X 0,Y 305.519,Z 265.428,A -85,B 0,C 180,E1 -15991.112,E2 -15991.112} C_VEL
LIN {X 0,Y 305.569,Z 265.423,A -85,B 0,C 180,E1 -15994.086,E2 -15994.086} C_VEL
LIN {X 0,Y 305.497,Z 265.433,A -85,B 0,C 180,E1 -15998.401,E2 -15998.401} C_VEL
LIN {X 0,Y 305.586,Z 265.421,A -85,B 0,C 180,E1 -16001.216,E2 -16001.216} C_VEL
LIN {X 0,Y 305.644,Z 265.414,A -85,B 0,C 180,E1 -16005.347,E2 -16005.347} C_VEL
LIN {X 0,Y 305.633,Z 265.416,A -85,B 0,C 180,E1 -16009.398,E2 -16009.398} C_VEL
LIN {X 0,Y 305.807,Z 265.394,A -85,B 0,C 180,E1 -16012.073,E2 -16012.073} C_VEL
LIN {X 0,Y 305.684,Z 265.406,A -85,B 0,C 180,E1 -16014.722,E2 -16014.722} C_VEL
LIN {X 0,Y 305.951,Z 265.375,A -85,B 0,C 180,E1 -16018.682,E2 -16018.682} C_VEL
LIN {X 0,Y 305.952,Z 265.376,A -85,B 0,C 180,E1 -16021.315,E2 -16021.315} C_VEL
LIN {X 0,Y 306.058,Z 267.851,A -85,B 0,C 180,E1 -16025.269,E2 -16025.269} C_VEL
LIN {X 0,Y 306.328,Z 269.686,A -85,B 0,C 180,E1 -16027.911,E2 -16027.911} C_VEL
LIN {X 0,Y 306.233,Z 271.728,A -85,B 0,C 180,E1 -16030.578,E2 -16030.578} C_VEL
LIN {X 0,Y 305.819,Z 275.124,A -85,B 0,C 180,E1 -16034.641,E2 -16034.641} C_VEL
LIN {X 0,Y 305.304,Z 278.86,A -85,B 0,C 180,E1 -16038.799,E2 -16038.799} C_VEL
LIN {X 0,Y 305.1,Z 280.456,A -85,B 0,C 180,E1 -16040.344,E2 -16040.344} C_VEL
LIN {X 0,Y 306.196,Z 283.623,A -85,B 0,C 180,E1 -16040.619,E2 -16040.619} C_VEL
LIN {X 0,Y 310.43,Z 295.737,A -85,B 0,C 180,E1 -16041.806,E2 -16041.806} C_VEL
LIN {X 0,Y 313.316,Z 306.92,A -85,B 0,C 180,E1 -16042.989,E2 -16042.989} C_VEL
LIN {X 0,Y 315.263,Z 318.532,A -85,B 0,C 180,E1 -16044.354,E2 -16044.354} C_VEL
LIN {X 0,Y 315.051,Z 321.854,A -85,B 0,C 180,E1 -16044.723,E2 -16044.723} C_VEL
LIN {X 0,Y 313.362,Z 332.66,A -85,B 0,C 180,E1 -16046.031,E2 -16046.031} C_VEL
LIN {X 0,Y 311.579,Z 342.649,A -85,B 0,C 180,E1 -16047.54,E2 -16047.54} C_VEL
LIN {X 0,Y 309.915,Z 351.439,A -85,B 0,C 180,E1 -16049.178,E2 -16049.178} C_VEL
LIN {X 0,Y 308.466,Z 358.883,A -85,B 0,C 180,E1 -16050.87,E2 -16050.87} C_VEL
LIN {X 0,Y 307.016,Z 365.626,A -85,B 0,C 180,E1 -16052.743,E2 -16052.743} C_VEL
LIN {X 0,Y 305.941,Z 371.022,A -85,B 0,C 180,E1 -16054.616,E2 -16054.616} C_VEL
LIN {X 0,Y 304.957,Z 375.945,A -85,B 0,C 180,E1 -16056.81,E2 -16056.81} C_VEL
LIN {X 0,Y 304.397,Z 378.93,A -85,B 0,C 180,E1 -16058.561,E2 -16058.561} C_VEL
LIN {X 0,Y 303.896,Z 381.174,A -85,B 0,C 180,E1 -16060.354,E2 -16060.354} C_VEL
LIN {X 0,Y 303.584,Z 382.708,A -85,B 0,C 180,E1 -16062.202,E2 -16062.202} C_VEL
LIN {X 0,Y 303.384,Z 383.485,A -85,B 0,C 180,E1 -16064.102,E2 -16064.102} C_VEL
LIN {X 0,Y 303.299,Z 383.44,A -85,B 0,C 180,E1 -16065.962,E2 -16065.962} C_VEL
LIN {X 0,Y 303.339,Z 382.578,A -85,B 0,C 180,E1 -16067.848,E2 -16067.848} C_VEL
LIN {X 0,Y 303.472,Z 380.792,A -85,B 0,C 180,E1 -16069.836,E2 -16069.836} C_VEL
LIN {X 0,Y 303.862,Z 378.015,A -85,B 0,C 180,E1 -16071.845,E2 -16071.845} C_VEL
LIN {X 0,Y 304.303,Z 374.027,A -85,B 0,C 180,E1 -16073.93,E2 -16073.93} C_VEL
LIN {X 0,Y 304.926,Z 368.642,A -85,B 0,C 180,E1 -16076.068,E2 -16076.068} C_VEL
LIN {X 0,Y 305.839,Z 361.606,A -85,B 0,C 180,E1 -16078.234,E2 -16078.234} C_VEL
LIN {X 0,Y 306.872,Z 353.878,A -85,B 0,C 180,E1 -16080.124,E2 -16080.124} C_VEL
LIN {X 0,Y 308.141,Z 344.121,A -85,B 0,C 180,E1 -16082.048,E2 -16082.048} C_VEL
LIN {X 0,Y 309.417,Z 333.472,A -85,B 0,C 180,E1 -16083.711,E2 -16083.711} C_VEL
LIN {X 0,Y 310.734,Z 322.554,A -85,B 0,C 180,E1 -16085.071,E2 -16085.071} C_VEL
LIN {X 0,Y 311.482,Z 314.862,A -85,B 0,C 180,E1 -16085.861,E2 -16085.861} C_VEL
LIN {X 0,Y 309.78,Z 303.491,A -85,B 0,C 180,E1 -16086.966,E2 -16086.966} C_VEL
LIN {X 0,Y 307.072,Z 290.233,A -85,B 0,C 180,E1 -16088.017,E2 -16088.017} C_VEL
LIN {X 0,Y 304.359,Z 278.813,A -85,B 0,C 180,E1 -16088.718,E2 -16088.718} C_VEL
LIN {X 0,Y 304.669,Z 274.675,A -85,B 0,C 180,E1 -16092.55,E2 -16092.55} C_VEL
LIN {X 0,Y 305.046,Z 270.343,A -85,B 0,C 180,E1 -16096.68,E2 -16096.68} C_VEL
LIN {X 0,Y 305.419,Z 266.212,A -85,B 0,C 180,E1 -16100.731,E2 -16100.731} C_VEL
LIN {X 0,Y 305.568,Z 265.421,A -85,B 0,C 180,E1 -16101.658,E2 -16101.658} C_VEL
LIN {X 0,Y 305.742,Z 265.398,A -85,B 0,C 180,E1 -16103.401,E2 -16103.401} C_VEL
LIN {X 0,Y 305.876,Z 265.381,A -85,B 0,C 180,E1 -16107.366,E2 -16107.366} C_VEL
LIN {X 0,Y 306.063,Z 265.359,A -85,B 0,C 180,E1 -16110,E2 -16110} C_VEL
LIN {X 0,Y 305.889,Z 265.383,A -85,B 0,C 180,E1 -16112.634,E2 -16112.634} C_VEL
LIN {X 0,Y 305.842,Z 265.389,A -85,B 0,C 180,E1 -16116.598,E2 -16116.598} C_VEL
LIN {X 0,Y 305.726,Z 265.4,A -85,B 0,C 180,E1 -16119.26,E2 -16119.26} C_VEL
LIN {X 0,Y 305.581,Z 265.418,A -85,B 0,C 180,E1 -16123.296,E2 -16123.296} C_VEL
LIN {X 0,Y 305.584,Z 265.422,A -85,B 0,C 180,E1 -16126.02,E2 -16126.02} C_VEL
LIN {X 0,Y 305.571,Z 265.419,A -85,B 0,C 180,E1 -16129.448,E2 -16129.448} C_VEL
LIN {X 0,Y 305.498,Z 265.428,A -85,B 0,C 180,E1 -16133.05,E2 -16133.05} C_VEL
LIN {X 0,Y 305.538,Z 265.424,A -85,B 0,C 180,E1 -16136.228,E2 -16136.228} C_VEL
LIN {X 0,Y 305.486,Z 265.428,A -85,B 0,C 180,E1 -16139.051,E2 -16139.051} C_VEL
LIN {X 0,Y 305.438,Z 265.439,A -85,B 0,C 180,E1 -16141.952,E2 -16141.952} C_VEL
LIN {X 0,Y 305.453,Z 265.435,A -85,B 0,C 180,E1 -16145.114,E2 -16145.114} C_VEL
LIN {X 0,Y 305.484,Z 265.429,A -85,B 0,C 180,E1 -16148.54,E2 -16148.54} C_VEL
LIN {X 0,Y 305.512,Z 265.424,A -85,B 0,C 180,E1 -16152.6,E2 -16152.6} C_VEL
LIN {X 0,Y 305.524,Z 265.424,A -85,B 0,C 180,E1 -16156.365,E2 -16156.365} C_VEL
LIN {X 0,Y 305.476,Z 265.432,A -85,B 0,C 180,E1 -16159.898,E2 -16159.898} C_VEL
LIN {X 0,Y 305.491,Z 265.43,A -85,B 0,C 180,E1 -16163.628,E2 -16163.628} C_VEL
LIN {X 0,Y 305.456,Z 265.432,A -85,B 0,C 180,E1 -16166.484,E2 -16166.484} C_VEL
LIN {X 0,Y 305.488,Z 265.431,A -85,B 0,C 180,E1 -16170.951,E2 -16170.951} C_VEL
LIN {X 0,Y 305.563,Z 265.419,A -85,B 0,C 180,E1 -16174.089,E2 -16174.089} C_VEL
LIN {X 0,Y 305.493,Z 265.431,A -85,B 0,C 180,E1 -16178.404,E2 -16178.404} C_VEL
LIN {X 0,Y 305.58,Z 265.418,A -85,B 0,C 180,E1 -16181.264,E2 -16181.264} C_VEL
LIN {X 0,Y 305.642,Z 265.408,A -85,B 0,C 180,E1 -16185.35,E2 -16185.35} C_VEL
LIN {X 0,Y 305.571,Z 265.417,A -85,B 0,C 180,E1 -16187.005,E2 -16187.005} C_VEL
LIN {X 0,Y 304.903,Z 265.502,A -85,B 0,C 180,E1 -16188.106,E2 -16188.106} C_VEL
LIN {X 0,Y 302.106,Z 265.848,A -85,B 0,C 180,E1 -16189.902,E2 -16189.902} C_VEL
LIN {X 0,Y 299.771,Z 266.14,A -85,B 0,C 180,E1 -16191.358,E2 -16191.358} C_VEL
LIN {X 0,Y 298.809,Z 266.265,A -85,B 0,C 180,E1 -16192.484,E2 -16192.484} C_VEL
LIN {X 0,Y 298.752,Z 266.266,A -85,B 0,C 180,E1 -16192.865,E2 -16192.865} C_VEL
LIN {X 0,Y 298.832,Z 266.258,A -85,B 0,C 180,E1 -16197.306,E2 -16197.306} C_VEL
LIN {X 0,Y 299.005,Z 266.24,A -85,B 0,C 180,E1 -16200.002,E2 -16200.002} C_VEL
LIN {X 0,Y 298.833,Z 266.257,A -85,B 0,C 180,E1 -16202.698,E2 -16202.698} C_VEL
LIN {X 0,Y 298.794,Z 266.262,A -85,B 0,C 180,E1 -16206.756,E2 -16206.756} C_VEL
LIN {X 0,Y 298.678,Z 266.278,A -85,B 0,C 180,E1 -16209.482,E2 -16209.482} C_VEL
LIN {X 0,Y 298.551,Z 266.296,A -85,B 0,C 180,E1 -16213.617,E2 -16213.617} C_VEL
LIN {X 0,Y 298.547,Z 266.293,A -85,B 0,C 180,E1 -16216.41,E2 -16216.41} C_VEL
LIN {X 0,Y 298.51,Z 266.301,A -85,B 0,C 180,E1 -16219.656,E2 -16219.656} C_VEL
LIN {X 0,Y 298.457,Z 266.31,A -85,B 0,C 180,E1 -16223.599,E2 -16223.599} C_VEL
LIN {X 0,Y 298.485,Z 266.301,A -85,B 0,C 180,E1 -16226.576,E2 -16226.576} C_VEL
LIN {X 0,Y 298.416,Z 266.314,A -85,B 0,C 180,E1 -16229.643,E2 -16229.643} C_VEL
LIN {X 0,Y 298.395,Z 266.314,A -85,B 0,C 180,E1 -16232.802,E2 -16232.802} C_VEL
LIN {X 0,Y 298.448,Z 266.308,A -85,B 0,C 180,E1 -16236.809,E2 -16236.809} C_VEL
LIN {X 0,Y 298.389,Z 266.318,A -85,B 0,C 180,E1 -16241.089,E2 -16241.089} C_VEL
LIN {X 0,Y 298.401,Z 266.317,A -85,B 0,C 180,E1 -16243.105,E2 -16243.105} C_VEL
LIN {X 0,Y 298.405,Z 266.389,A -85,B 0,C 180,E1 -16245.918,E2 -16245.918} C_VEL
LIN {X 0,Y 299.256,Z 270.967,A -85,B 0,C 180,E1 -16249.772,E2 -16249.772} C_VEL
LIN {X 0,Y 299.702,Z 274.292,A -85,B 0,C 180,E1 -16252.433,E2 -16252.433} C_VEL
LIN {X 0,Y 299.792,Z 277.827,A -85,B 0,C 180,E1 -16255.137,E2 -16255.137} C_VEL
LIN {X 0,Y 298.967,Z 282.957,A -85,B 0,C 180,E1 -16258.858,E2 -16258.858} C_VEL
LIN {X 0,Y 298.117,Z 289.689,A -85,B 0,C 180,E1 -16263.619,E2 -16263.619} C_VEL
LIN {X 0,Y 297.716,Z 294.511,A -85,B 0,C 180,E1 -16266.875,E2 -16266.875} C_VEL
LIN {X 0,Y 300.211,Z 308,A -85,B 0,C 180,E1 -16267.664,E2 -16267.664} C_VEL
LIN {X 0,Y 302.073,Z 321.141,A -85,B 0,C 180,E1 -16268.686,E2 -16268.686} C_VEL
LIN {X 0,Y 303.211,Z 331.165,A -85,B 0,C 180,E1 -16269.655,E2 -16269.655} C_VEL
LIN {X 0,Y 303.621,Z 337.817,A -85,B 0,C 180,E1 -16270.389,E2 -16270.389} C_VEL
LIN {X 0,Y 302.165,Z 348.575,A -85,B 0,C 180,E1 -16271.7,E2 -16271.7} C_VEL
LIN {X 0,Y 300.79,Z 359.175,A -85,B 0,C 180,E1 -16273.333,E2 -16273.333} C_VEL
LIN {X 0,Y 299.633,Z 368.18,A -85,B 0,C 180,E1 -16275.048,E2 -16275.048} C_VEL
LIN {X 0,Y 298.637,Z 375.454,A -85,B 0,C 180,E1 -16276.735,E2 -16276.735} C_VEL
LIN {X 0,Y 297.705,Z 382.6,A -85,B 0,C 180,E1 -16278.769,E2 -16278.769} C_VEL
LIN {X 0,Y 297.044,Z 389.108,A -85,B 0,C 180,E1 -16281.153,E2 -16281.153} C_VEL
LIN {X 0,Y 296.696,Z 393.384,A -85,B 0,C 180,E1 -16283.198,E2 -16283.198} C_VEL
LIN {X 0,Y 296.557,Z 395.641,A -85,B 0,C 180,E1 -16284.56,E2 -16284.56} C_VEL
LIN {X 0,Y 296.533,Z 397.417,A -85,B 0,C 180,E1 -16285.923,E2 -16285.923} C_VEL
LIN {X 0,Y 296.537,Z 398.75,A -85,B 0,C 180,E1 -16287.283,E2 -16287.283} C_VEL
LIN {X 0,Y 296.497,Z 399.677,A -85,B 0,C 180,E1 -16288.642,E2 -16288.642} C_VEL
LIN {X 0,Y 296.521,Z 400.207,A -85,B 0,C 180,E1 -16290,E2 -16290} C_VEL
LIN {X 0,Y 296.487,Z 400.294,A -85,B 0,C 180,E1 -16291.358,E2 -16291.358} C_VEL
LIN {X 0,Y 296.529,Z 399.98,A -85,B 0,C 180,E1 -16292.717,E2 -16292.717} C_VEL
LIN {X 0,Y 296.537,Z 398.18,A -85,B 0,C 180,E1 -16295.44,E2 -16295.44} C_VEL
LIN {X 0,Y 296.692,Z 396.64,A -85,B 0,C 180,E1 -16296.802,E2 -16296.802} C_VEL
LIN {X 0,Y 297.127,Z 393.543,A -85,B 0,C 180,E1 -16298.844,E2 -16298.844} C_VEL
LIN {X 0,Y 297.776,Z 389.404,A -85,B 0,C 180,E1 -16300.883,E2 -16300.883} C_VEL
LIN {X 0,Y 298.927,Z 383.099,A -85,B 0,C 180,E1 -16303.251,E2 -16303.251} C_VEL
LIN {X 0,Y 300.448,Z 376.29,A -85,B 0,C 180,E1 -16305.257,E2 -16305.257} C_VEL
LIN {X 0,Y 301.889,Z 368.351,A -85,B 0,C 180,E1 -16307.168,E2 -16307.168} C_VEL
LIN {X 0,Y 303.647,Z 359.351,A -85,B 0,C 180,E1 -16308.906,E2 -16308.906} C_VEL
LIN {X 0,Y 305.719,Z 348.9,A -85,B 0,C 180,E1 -16310.522,E2 -16310.522} C_VEL
LIN {X 0,Y 307.113,Z 340.215,A -85,B 0,C 180,E1 -16311.633,E2 -16311.633} C_VEL
LIN {X 0,Y 306.61,Z 329.629,A -85,B 0,C 180,E1 -16312.933,E2 -16312.933} C_VEL
LIN {X 0,Y 305.098,Z 318.188,A -85,B 0,C 180,E1 -16314.186,E2 -16314.186} C_VEL
LIN {X 0,Y 302.803,Z 307.611,A -85,B 0,C 180,E1 -16315.238,E2 -16315.238} C_VEL
LIN {X 0,Y 299.27,Z 295.939,A -85,B 0,C 180,E1 -16316.31,E2 -16316.31} C_VEL
LIN {X 0,Y 298.491,Z 292.881,A -85,B 0,C 180,E1 -16316.573,E2 -16316.573} C_VEL
LIN {X 0,Y 299.071,Z 288.881,A -85,B 0,C 180,E1 -16319.6,E2 -16319.6} C_VEL
LIN {X 0,Y 299.686,Z 285.01,A -85,B 0,C 180,E1 -16322.64,E2 -16322.64} C_VEL
LIN {X 0,Y 300.214,Z 281.19,A -85,B 0,C 180,E1 -16325.82,E2 -16325.82} C_VEL
LIN {X 0,Y 300.305,Z 279.323,A -85,B 0,C 180,E1 -16327.478,E2 -16327.478} C_VEL
LIN {X 0,Y 299.961,Z 275.707,A -85,B 0,C 180,E1 -16330.997,E2 -16330.997} C_VEL
LIN {X 0,Y 299.429,Z 272.257,A -85,B 0,C 180,E1 -16334.759,E2 -16334.759} C_VEL
LIN {X 0,Y 298.901,Z 269.005,A -85,B 0,C 180,E1 -16338.824,E2 -16338.824} C_VEL
LIN {X 0,Y 298.48,Z 266.685,A -85,B 0,C 180,E1 -16342.25,E2 -16342.25} C_VEL
LIN {X 0,Y 298.431,Z 266.313,A -85,B 0,C 180,E1 -16343.93,E2 -16343.93} C_VEL
LIN {X 0,Y 298.394,Z 266.317,A -85,B 0,C 180,E1 -16347.982,E2 -16347.982} C_VEL
LIN {X 0,Y 298.462,Z 266.308,A -85,B 0,C 180,E1 -16351.903,E2 -16351.903} C_VEL
LIN {X 0,Y 298.483,Z 266.305,A -85,B 0,C 180,E1 -16354.922,E2 -16354.922} C_VEL
LIN {X 0,Y 298.446,Z 266.312,A -85,B 0,C 180,E1 -16359.314,E2 -16359.314} C_VEL
LIN {X 0,Y 298.534,Z 266.3,A -85,B 0,C 180,E1 -16362.178,E2 -16362.178} C_VEL
LIN {X 0,Y 298.589,Z 266.293,A -85,B 0,C 180,E1 -16364.993,E2 -16364.993} C_VEL
LIN {X 0,Y 298.589,Z 266.293,A -85,B 0,C 180,E1 -16369.145,E2 -16369.145} C_VEL
LIN {X 0,Y 298.753,Z 266.273,A -85,B 0,C 180,E1 -16371.884,E2 -16371.884} C_VEL
LIN {X 0,Y 298.655,Z 266.282,A -85,B 0,C 180,E1 -16374.597,E2 -16374.597} C_VEL
LIN {X 0,Y 298.917,Z 266.25,A -85,B 0,C 180,E1 -16378.651,E2 -16378.651} C_VEL
LIN {X 0,Y 299.003,Z 266.24,A -85,B 0,C 180,E1 -16379.998,E2 -16379.998} C_VEL
LIN {X 0,Y 299.043,Z 267.567,A -85,B 0,C 180,E1 -16382.692,E2 -16382.692} C_VEL
LIN {X 0,Y 299.252,Z 270.231,A -85,B 0,C 180,E1 -16386.832,E2 -16386.832} C_VEL
LIN {X 0,Y 299.34,Z 272.188,A -85,B 0,C 180,E1 -16389.576,E2 -16389.576} C_VEL
LIN {X 0,Y 298.889,Z 275.401,A -85,B 0,C 180,E1 -16393.598,E2 -16393.598} C_VEL
LIN {X 0,Y 298.52,Z 277.793,A -85,B 0,C 180,E1 -16396.408,E2 -16396.408} C_VEL
LIN {X 0,Y 298.178,Z 280.683,A -85,B 0,C 180,E1 -16399.516,E2 -16399.516} C_VEL
LIN {X 0,Y 299.207,Z 283.756,A -85,B 0,C 180,E1 -16399.795,E2 -16399.795} C_VEL
LIN {X 0,Y 303.099,Z 294.327,A -85,B 0,C 180,E1 -16400.884,E2 -16400.884} C_VEL
LIN {X 0,Y 305.999,Z 304.546,A -85,B 0,C 180,E1 -16402.01,E2 -16402.01} C_VEL
LIN {X 0,Y 308.223,Z 316.069,A -85,B 0,C 180,E1 -16403.391,E2 -16403.391} C_VEL
LIN {X 0,Y 308.811,Z 321.283,A -85,B 0,C 180,E1 -16404.056,E2 -16404.056} C_VEL
LIN {X 0,Y 306.994,Z 332.499,A -85,B 0,C 180,E1 -16405.417,E2 -16405.417} C_VEL
LIN {X 0,Y 305.237,Z 341.924,A -85,B 0,C 180,E1 -16406.846,E2 -16406.846} C_VEL
LIN {X 0,Y 303.227,Z 351.875,A -85,B 0,C 180,E1 -16408.721,E2 -16408.721} C_VEL
LIN {X 0,Y 301.695,Z 359.34,A -85,B 0,C 180,E1 -16410.47,E2 -16410.47} C_VEL
LIN {X 0,Y 300.024,Z 366.664,A -85,B 0,C 180,E1 -16412.598,E2 -16412.598} C_VEL
LIN {X 0,Y 298.843,Z 372.105,A -85,B 0,C 180,E1 -16414.605,E2 -16414.605} C_VEL
LIN {X 0,Y 297.936,Z 376.497,A -85,B 0,C 180,E1 -16416.678,E2 -16416.678} C_VEL
